LIN {X 0,Y 161.078,Z 235.028,A -85,B 0,C 180,E1 -25523.5,E2 -25523.5} C_VEL
LIN {X 0,Y 155.876,Z 225.999,A -85,B 0,C 180,E1 -25526.938,E2 -25526.938} C_VEL
LIN {X 0,Y 150.877,Z 218.256,A -85,B 0,C 180,E1 -25530.745,E2 -25530.745} C_VEL
LIN {X 0,Y 148.583,Z 214.919,A -85,B 0,C 180,E1 -25532.727,E2 -25532.727} C_VEL
LIN {X 0,Y 145.779,Z 210.989,A -85,B 0,C 180,E1 -25535.429,E2 -25535.429} C_VEL
LIN {X 0,Y 142.918,Z 207.15,A -85,B 0,C 180,E1 -25538.623,E2 -25538.623} C_VEL
LIN {X 0,Y 142.606,Z 206.481,A -85,B 0,C 180,E1 -25539.043,E2 -25539.043} C_VEL
LIN {X 0,Y 140.021,Z 203.936,A -85,B 0,C 180,E1 -25542.473,E2 -25542.473} C_VEL
LIN {X 0,Y 138.637,Z 201.246,A -85,B 0,C 180,E1 -25544.941,E2 -25544.941} C_VEL
LIN {X 0,Y 135.796,Z 198.706,A -85,B 0,C 180,E1 -25551.349,E2 -25551.349} C_VEL
LIN {X 0,Y 134.805,Z 195.544,A -85,B 0,C 180,E1 -25557.759,E2 -25557.759} C_VEL
LIN {X 0,Y 134.795,Z 195.447,A -85,B 0,C 180,E1 -25561.494,E2 -25561.494} C_VEL
LIN {X 0,Y 134.949,Z 196.715,A -85,B 0,C 180,E1 -25564.013,E2 -25564.013} C_VEL
LIN {X 0,Y 137.876,Z 200.864,A -85,B 0,C 180,E1 -25573.261,E2 -25573.261} C_VEL
LIN {X 0,Y 138.78,Z 201.463,A -85,B 0,C 180,E1 -25574.855,E2 -25574.855} C_VEL
LIN {X 0,Y 140.657,Z 204.791,A -85,B 0,C 180,E1 -25578.009,E2 -25578.009} C_VEL
LIN {X 0,Y 142.764,Z 206.915,A -85,B 0,C 180,E1 -25580.716,E2 -25580.716} C_VEL
LIN {X 0,Y 145.209,Z 210.44,A -85,B 0,C 180,E1 -25583.534,E2 -25583.534} C_VEL
LIN {X 0,Y 146.412,Z 211.841,A -85,B 0,C 180,E1 -25584.741,E2 -25584.741} C_VEL
LIN {X 0,Y 149.716,Z 216.584,A -85,B 0,C 180,E1 -25587.808,E2 -25587.808} C_VEL
LIN {X 0,Y 152.19,Z 220.352,A -85,B 0,C 180,E1 -25589.859,E2 -25589.859} C_VEL
LIN {X 0,Y 156.704,Z 229.259,A -85,B 0,C 180,E1 -25593.326,E2 -25593.326} C_VEL
LIN {X 0,Y 161.77,Z 240.791,A -85,B 0,C 180,E1 -25596.782,E2 -25596.782} C_VEL
LIN {X 0,Y 165.726,Z 251.888,A -85,B 0,C 180,E1 -25599.306,E2 -25599.306} C_VEL
LIN {X 0,Y 165.659,Z 255.549,A -85,B 0,C 180,E1 -25599.521,E2 -25599.521} C_VEL
LIN {X 0,Y 163.102,Z 287.628,A -85,B 0,C 180,E1 -25600.707,E2 -25600.707} C_VEL
LIN {X 0,Y 160.961,Z 301.09,A -85,B 0,C 180,E1 -25601.558,E2 -25601.558} C_VEL
LIN {X 0,Y 157.935,Z 313.779,A -85,B 0,C 180,E1 -25602.756,E2 -25602.756} C_VEL
LIN {X 0,Y 154.381,Z 324.846,A -85,B 0,C 180,E1 -25604.192,E2 -25604.192} C_VEL
LIN {X 0,Y 149.882,Z 336.398,A -85,B 0,C 180,E1 -25606.24,E2 -25606.24} C_VEL
LIN {X 0,Y 145.19,Z 346.81,A -85,B 0,C 180,E1 -25608.735,E2 -25608.735} C_VEL
LIN {X 0,Y 140.727,Z 355.322,A -85,B 0,C 180,E1 -25611.371,E2 -25611.371} C_VEL
LIN {X 0,Y 136.248,Z 363.183,A -85,B 0,C 180,E1 -25614.527,E2 -25614.527} C_VEL
LIN {X 0,Y 132.327,Z 369.715,A -85,B 0,C 180,E1 -25617.918,E2 -25617.918} C_VEL
LIN {X 0,Y 128.273,Z 376.146,A -85,B 0,C 180,E1 -25622.242,E2 -25622.242} C_VEL
LIN {X 0,Y 124.805,Z 381.256,A -85,B 0,C 180,E1 -25626.784,E2 -25626.784} C_VEL
LIN {X 0,Y 122.116,Z 385.23,A -85,B 0,C 180,E1 -25631.545,E2 -25631.545} C_VEL
LIN {X 0,Y 120.445,Z 388.179,A -85,B 0,C 180,E1 -25636.501,E2 -25636.501} C_VEL
LIN {X 0,Y 119.32,Z 390.59,A -85,B 0,C 180,E1 -25643.233,E2 -25643.233} C_VEL
LIN {X 0,Y 119.284,Z 391.21,A -85,B 0,C 180,E1 -25646.621,E2 -25646.621} C_VEL
LIN {X 0,Y 119.417,Z 391.429,A -85,B 0,C 180,E1 -25649.998,E2 -25649.998} C_VEL
LIN {X 0,Y 119.284,Z 391.193,A -85,B 0,C 180,E1 -25653.376,E2 -25653.376} C_VEL
LIN {X 0,Y 119.382,Z 390.566,A -85,B 0,C 180,E1 -25656.76,E2 -25656.76} C_VEL
LIN {X 0,Y 120.446,Z 388.126,A -85,B 0,C 180,E1 -25663.495,E2 -25663.495} C_VEL
LIN {X 0,Y 122.113,Z 385.154,A -85,B 0,C 180,E1 -25668.452,E2 -25668.452} C_VEL
LIN {X 0,Y 125.137,Z 380.624,A -85,B 0,C 180,E1 -25673.724,E2 -25673.724} C_VEL
LIN {X 0,Y 128.93,Z 375.007,A -85,B 0,C 180,E1 -25678.485,E2 -25678.485} C_VEL
LIN {X 0,Y 133.088,Z 368.298,A -85,B 0,C 180,E1 -25682.768,E2 -25682.768} C_VEL
LIN {X 0,Y 135.059,Z 364.976,A -85,B 0,C 180,E1 -25684.506,E2 -25684.506} C_VEL
LIN {X 0,Y 136.621,Z 361.327,A -85,B 0,C 180,E1 -25686.354,E2 -25686.354} C_VEL
LIN {X 0,Y 137.849,Z 355.051,A -85,B 0,C 180,E1 -25689.523,E2 -25689.523} C_VEL
LIN {X 0,Y 139.287,Z 348.297,A -85,B 0,C 180,E1 -25692.442,E2 -25692.442} C_VEL
LIN {X 0,Y 141.091,Z 343.81,A -85,B 0,C 180,E1 -25693.844,E2 -25693.844} C_VEL
LIN {X 0,Y 145.975,Z 333.133,A -85,B 0,C 180,E1 -25696.232,E2 -25696.232} C_VEL
LIN {X 0,Y 150.71,Z 320.63,A -85,B 0,C 180,E1 -25698.252,E2 -25698.252} C_VEL
LIN {X 0,Y 154.39,Z 308.335,A -85,B 0,C 180,E1 -25699.68,E2 -25699.68} C_VEL
LIN {X 0,Y 157.155,Z 295.303,A -85,B 0,C 180,E1 -25700.732,E2 -25700.732} C_VEL
LIN {X 0,Y 158.826,Z 282.23,A -85,B 0,C 180,E1 -25701.429,E2 -25701.429} C_VEL
LIN {X 0,Y 161.036,Z 254.175,A -85,B 0,C 180,E1 -25702.437,E2 -25702.437} C_VEL
LIN {X 0,Y 157.36,Z 243.724,A -85,B 0,C 180,E1 -25704.996,E2 -25704.996} C_VEL
LIN {X 0,Y 152.664,Z 232.741,A -85,B 0,C 180,E1 -25708.519,E2 -25708.519} C_VEL
LIN {X 0,Y 148.861,Z 224.979,A -85,B 0,C 180,E1 -25711.726,E2 -25711.726} C_VEL
LIN {X 0,Y 145.92,Z 220.592,A -85,B 0,C 180,E1 -25714.408,E2 -25714.408} C_VEL
LIN {X 0,Y 143.478,Z 217.065,A -85,B 0,C 180,E1 -25716.93,E2 -25716.93} C_VEL
LIN {X 0,Y 140.56,Z 212.9,A -85,B 0,C 180,E1 -25720.466,E2 -25720.466} C_VEL
LIN {X 0,Y 137.986,Z 209.737,A -85,B 0,C 180,E1 -25724.259,E2 -25724.259} C_VEL
LIN {X 0,Y 137.127,Z 208.03,A -85,B 0,C 180,E1 -25725.91,E2 -25725.91} C_VEL
LIN {X 0,Y 134.691,Z 205.604,A -85,B 0,C 180,E1 -25731.561,E2 -25731.561} C_VEL
LIN {X 0,Y 133.728,Z 202.571,A -85,B 0,C 180,E1 -25736.988,E2 -25736.988} C_VEL
LIN {X 0,Y 133.536,Z 202.368,A -85,B 0,C 180,E1 -25740.678,E2 -25740.678} C_VEL
LIN {X 0,Y 133.734,Z 202.746,A -85,B 0,C 180,E1 -25743.767,E2 -25743.767} C_VEL
LIN {X 0,Y 135.902,Z 207.202,A -85,B 0,C 180,E1 -25752.266,E2 -25752.266} C_VEL
LIN {X 0,Y 137.366,Z 208.395,A -85,B 0,C 180,E1 -25755.106,E2 -25755.106} C_VEL
LIN {X 0,Y 139.567,Z 211.978,A -85,B 0,C 180,E1 -25758.783,E2 -25758.783} C_VEL
LIN {X 0,Y 141.064,Z 213.572,A -85,B 0,C 180,E1 -25760.749,E2 -25760.749} C_VEL
LIN {X 0,Y 143.805,Z 217.401,A -85,B 0,C 180,E1 -25763.97,E2 -25763.97} C_VEL
LIN {X 0,Y 147.63,Z 223.134,A -85,B 0,C 180,E1 -25767.752,E2 -25767.752} C_VEL
LIN {X 0,Y 152.022,Z 230.155,A -85,B 0,C 180,E1 -25771.417,E2 -25771.417} C_VEL
LIN {X 0,Y 156.705,Z 238.412,A -85,B 0,C 180,E1 -25774.804,E2 -25774.804} C_VEL
LIN {X 0,Y 161.45,Z 247.957,A -85,B 0,C 180,E1 -25777.868,E2 -25777.868} C_VEL
LIN {X 0,Y 159.713,Z 271.663,A -85,B 0,C 180,E1 -25778.762,E2 -25778.762} C_VEL
LIN {X 0,Y 158.229,Z 285.038,A -85,B 0,C 180,E1 -25779.38,E2 -25779.38} C_VEL
LIN {X 0,Y 155.784,Z 298.21,A -85,B 0,C 180,E1 -25780.425,E2 -25780.425} C_VEL
LIN {X 0,Y 152.866,Z 309.358,A -85,B 0,C 180,E1 -25781.664,E2 -25781.664} C_VEL
LIN {X 0,Y 148.975,Z 321.287,A -85,B 0,C 180,E1 -25783.507,E2 -25783.507} C_VEL
LIN {X 0,Y 144.587,Z 331.921,A -85,B 0,C 180,E1 -25785.678,E2 -25785.678} C_VEL
LIN {X 0,Y 139.895,Z 341.613,A -85,B 0,C 180,E1 -25788.271,E2 -25788.271} C_VEL
LIN {X 0,Y 135.201,Z 350.422,A -85,B 0,C 180,E1 -25791.41,E2 -25791.41} C_VEL
LIN {X 0,Y 129.901,Z 359.017,A -85,B 0,C 180,E1 -25795.386,E2 -25795.386} C_VEL
LIN {X 0,Y 125.108,Z 365.872,A -85,B 0,C 180,E1 -25799.633,E2 -25799.633} C_VEL
LIN {X 0,Y 121.098,Z 371.353,A -85,B 0,C 180,E1 -25804.2,E2 -25804.2} C_VEL
LIN {X 0,Y 117.817,Z 375.652,A -85,B 0,C 180,E1 -25809.03,E2 -25809.03} C_VEL
LIN {X 0,Y 116.068,Z 377.924,A -85,B 0,C 180,E1 -25812.379,E2 -25812.379} C_VEL
LIN {X 0,Y 114.679,Z 379.769,A -85,B 0,C 180,E1 -25815.812,E2 -25815.812} C_VEL
LIN {X 0,Y 113.654,Z 381.152,A -85,B 0,C 180,E1 -25819.311,E2 -25819.311} C_VEL
LIN {X 0,Y 112.553,Z 382.738,A -85,B 0,C 180,E1 -25826.422,E2 -25826.422} C_VEL
LIN {X 0,Y 112.46,Z 382.938,A -85,B 0,C 180,E1 -25830.807,E2 -25830.807} C_VEL
LIN {X 0,Y 112.937,Z 382.183,A -85,B 0,C 180,E1 -25837.151,E2 -25837.151} C_VEL
LIN {X 0,Y 113.652,Z 381.217,A -85,B 0,C 180,E1 -25840.693,E2 -25840.693} C_VEL
LIN {X 0,Y 114.63,Z 379.865,A -85,B 0,C 180,E1 -25844.198,E2 -25844.198} C_VEL
LIN {X 0,Y 116.865,Z 377,A -85,B 0,C 180,E1 -25849.316,E2 -25849.316} C_VEL
LIN {X 0,Y 119.883,Z 373.112,A -85,B 0,C 180,E1 -25854.229,E2 -25854.229} C_VEL
LIN {X 0,Y 123.638,Z 368.095,A -85,B 0,C 180,E1 -25858.894,E2 -25858.894} C_VEL
LIN {X 0,Y 128.178,Z 361.767,A -85,B 0,C 180,E1 -25863.252,E2 -25863.252} C_VEL
LIN {X 0,Y 133.004,Z 354.314,A -85,B 0,C 180,E1 -25867.125,E2 -25867.125} C_VEL
LIN {X 0,Y 137.799,Z 345.963,A -85,B 0,C 180,E1 -25870.467,E2 -25870.467} C_VEL
LIN {X 0,Y 142.911,Z 335.935,A -85,B 0,C 180,E1 -25873.512,E2 -25873.512} C_VEL
LIN {X 0,Y 147.779,Z 324.829,A -85,B 0,C 180,E1 -25875.998,E2 -25875.998} C_VEL
LIN {X 0,Y 151.697,Z 313.941,A -85,B 0,C 180,E1 -25877.841,E2 -25877.841} C_VEL
LIN {X 0,Y 155.184,Z 301.895,A -85,B 0,C 180,E1 -25879.34,E2 -25879.34} C_VEL
LIN {X 0,Y 157.827,Z 288.964,A -85,B 0,C 180,E1 -25880.506,E2 -25880.506} C_VEL
LIN {X 0,Y 159.598,Z 275.623,A -85,B 0,C 180,E1 -25881.23,E2 -25881.23} C_VEL
LIN {X 0,Y 161.694,Z 248.648,A -85,B 0,C 180,E1 -25882.22,E2 -25882.22} C_VEL
LIN {X 0,Y 160.961,Z 246.685,A -85,B 0,C 180,E1 -25882.703,E2 -25882.703} C_VEL
LIN {X 0,Y 156.156,Z 237.203,A -85,B 0,C 180,E1 -25885.863,E2 -25885.863} C_VEL
LIN {X 0,Y 151.23,Z 228.617,A -85,B 0,C 180,E1 -25889.533,E2 -25889.533} C_VEL
LIN {X 0,Y 146.854,Z 221.695,A -85,B 0,C 180,E1 -25893.342,E2 -25893.342} C_VEL
LIN {X 0,Y 143.607,Z 217.135,A -85,B 0,C 180,E1 -25896.644,E2 -25896.644} C_VEL
LIN {X 0,Y 140.638,Z 212.926,A -85,B 0,C 180,E1 -25900.286,E2 -25900.286} C_VEL
LIN {X 0,Y 138.04,Z 209.692,A -85,B 0,C 180,E1 -25904.213,E2 -25904.213} C_VEL
LIN {X 0,Y 137.279,Z 208.068,A -85,B 0,C 180,E1 -25905.737,E2 -25905.737} C_VEL
LIN {X 0,Y 134.732,Z 205.56,A -85,B 0,C 180,E1 -25911.988,E2 -25911.988} C_VEL
LIN {X 0,Y 133.9,Z 202.507,A -85,B 0,C 180,E1 -25918.496,E2 -25918.496} C_VEL
LIN {X 0,Y 133.931,Z 202.725,A -85,B 0,C 180,E1 -25921.879,E2 -25921.879} C_VEL
LIN {X 0,Y 135.58,Z 206.699,A -85,B 0,C 180,E1 -25930.165,E2 -25930.165} C_VEL
LIN {X 0,Y 137.455,Z 208.381,A -85,B 0,C 180,E1 -25934.15,E2 -25934.15} C_VEL
LIN {X 0,Y 139.436,Z 211.737,A -85,B 0,C 180,E1 -25937.603,E2 -25937.603} C_VEL
LIN {X 0,Y 141.019,Z 213.431,A -85,B 0,C 180,E1 -25939.752,E2 -25939.752} C_VEL
LIN {X 0,Y 143.578,Z 217.152,A -85,B 0,C 180,E1 -25942.863,E2 -25942.863} C_VEL
LIN {X 0,Y 144.8,Z 218.877,A -85,B 0,C 180,E1 -25944.175,E2 -25944.175} C_VEL
LIN {X 0,Y 147.706,Z 223.15,A -85,B 0,C 180,E1 -25946.999,E2 -25946.999} C_VEL
LIN {X 0,Y 149.699,Z 226.419,A -85,B 0,C 180,E1 -25948.765,E2 -25948.765} C_VEL
LIN {X 0,Y 154.034,Z 235.4,A -85,B 0,C 180,E1 -25952.322,E2 -25952.322} C_VEL
LIN {X 0,Y 158.785,Z 247.167,A -85,B 0,C 180,E1 -25955.812,E2 -25955.812} C_VEL
LIN {X 0,Y 161.231,Z 254.426,A -85,B 0,C 180,E1 -25957.51,E2 -25957.51} C_VEL
LIN {X 0,Y 158.542,Z 287.605,A -85,B 0,C 180,E1 -25958.777,E2 -25958.777} C_VEL
LIN {X 0,Y 156.413,Z 300.586,A -85,B 0,C 180,E1 -25959.601,E2 -25959.601} C_VEL
LIN {X 0,Y 153.212,Z 313.527,A -85,B 0,C 180,E1 -25960.81,E2 -25960.81} C_VEL
LIN {X 0,Y 149.522,Z 324.592,A -85,B 0,C 180,E1 -25962.242,E2 -25962.242} C_VEL
LIN {X 0,Y 144.836,Z 336.143,A -85,B 0,C 180,E1 -25964.296,E2 -25964.296} C_VEL
LIN {X 0,Y 139.914,Z 346.553,A -85,B 0,C 180,E1 -25966.811,E2 -25966.811} C_VEL
LIN {X 0,Y 135.25,Z 355.066,A -85,B 0,C 180,E1 -25969.492,E2 -25969.492} C_VEL
LIN {X 0,Y 129.627,Z 364.299,A -85,B 0,C 180,E1 -25973.387,E2 -25973.387} C_VEL
LIN {X 0,Y 124.582,Z 371.977,A -85,B 0,C 180,E1 -25977.8,E2 -25977.8} C_VEL
LIN {X 0,Y 120.634,Z 377.71,A -85,B 0,C 180,E1 -25982.219,E2 -25982.219} C_VEL
LIN {X 0,Y 117.215,Z 382.434,A -85,B 0,C 180,E1 -25987.061,E2 -25987.061} C_VEL
LIN {X 0,Y 114.629,Z 386.048,A -85,B 0,C 180,E1 -25992.147,E2 -25992.147} C_VEL
LIN {X 0,Y 113.503,Z 387.919,A -85,B 0,C 180,E1 -25995.658,E2 -25995.658} C_VEL
LIN {X 0,Y 112.708,Z 389.324,A -85,B 0,C 180,E1 -25999.217,E2 -25999.217} C_VEL
LIN {X 0,Y 112.177,Z 390.95,A -85,B 0,C 180,E1 -26006.406,E2 -26006.406} C_VEL
LIN {X 0,Y 112.332,Z 391.17,A -85,B 0,C 180,E1 -26009.998,E2 -26009.998} C_VEL
LIN {X 0,Y 112.2,Z 390.934,A -85,B 0,C 180,E1 -26013.589,E2 -26013.589} C_VEL
LIN {X 0,Y 112.304,Z 390.305,A -85,B 0,C 180,E1 -26017.188,E2 -26017.188} C_VEL
LIN {X 0,Y 112.728,Z 389.287,A -85,B 0,C 180,E1 -26020.778,E2 -26020.778} C_VEL
LIN {X 0,Y 113.504,Z 387.864,A -85,B 0,C 180,E1 -26024.338,E2 -26024.338} C_VEL
LIN {X 0,Y 115.377,Z 384.893,A -85,B 0,C 180,E1 -26029.572,E2 -26029.572} C_VEL
LIN {X 0,Y 118.291,Z 380.891,A -85,B 0,C 180,E1 -26034.573,E2 -26034.573} C_VEL
LIN {X 0,Y 122.693,Z 374.745,A -85,B 0,C 180,E1 -26040.078,E2 -26040.078} C_VEL
LIN {X 0,Y 127.145,Z 368.036,A -85,B 0,C 180,E1 -26044.509,E2 -26044.509} C_VEL
LIN {X 0,Y 132.34,Z 359.723,A -85,B 0,C 180,E1 -26048.605,E2 -26048.605} C_VEL
LIN {X 0,Y 137.263,Z 351.204,A -85,B 0,C 180,E1 -26051.726,E2 -26051.726} C_VEL
LIN {X 0,Y 141.091,Z 343.81,A -85,B 0,C 180,E1 -26053.844,E2 -26053.844} C_VEL
LIN {X 0,Y 142.876,Z 339.205,A -85,B 0,C 180,E1 -26055.161,E2 -26055.161} C_VEL
LIN {X 0,Y 144.301,Z 331.465,A -85,B 0,C 180,E1 -26057.581,E2 -26057.581} C_VEL
LIN {X 0,Y 145.524,Z 323.296,A -85,B 0,C 180,E1 -26059.747,E2 -26059.747} C_VEL
LIN {X 0,Y 146.901,Z 318.027,A -85,B 0,C 180,E1 -26060.637,E2 -26060.637} C_VEL
LIN {X 0,Y 150.529,Z 305.51,A -85,B 0,C 180,E1 -26061.984,E2 -26061.984} C_VEL
LIN {X 0,Y 153.293,Z 292.019,A -85,B 0,C 180,E1 -26062.979,E2 -26062.979} C_VEL
LIN {X 0,Y 154.814,Z 278.296,A -85,B 0,C 180,E1 -26063.631,E2 -26063.631} C_VEL
LIN {X 0,Y 156.594,Z 256.462,A -85,B 0,C 180,E1 -26064.406,E2 -26064.406} C_VEL
LIN {X 0,Y 153.415,Z 247.166,A -85,B 0,C 180,E1 -26066.848,E2 -26066.848} C_VEL
LIN {X 0,Y 149.09,Z 236.597,A -85,B 0,C 180,E1 -26070.444,E2 -26070.444} C_VEL
LIN {X 0,Y 146.018,Z 230.346,A -85,B 0,C 180,E1 -26073.274,E2 -26073.274} C_VEL
LIN {X 0,Y 143.656,Z 226.611,A -85,B 0,C 180,E1 -26075.62,E2 -26075.62} C_VEL
LIN {X 0,Y 141.562,Z 223.441,A -85,B 0,C 180,E1 -26077.948,E2 -26077.948} C_VEL
LIN {X 0,Y 138.794,Z 219.375,A -85,B 0,C 180,E1 -26081.55,E2 -26081.55} C_VEL
LIN {X 0,Y 136.395,Z 216.043,A -85,B 0,C 180,E1 -26085.452,E2 -26085.452} C_VEL
LIN {X 0,Y 135.883,Z 214.882,A -85,B 0,C 180,E1 -26086.541,E2 -26086.541} C_VEL
LIN {X 0,Y 133.605,Z 212.437,A -85,B 0,C 180,E1 -26092.253,E2 -26092.253} C_VEL
LIN {X 0,Y 132.783,Z 209.548,A -85,B 0,C 180,E1 -26097.725,E2 -26097.725} C_VEL
LIN {X 0,Y 132.801,Z 209.574,A -85,B 0,C 180,E1 -26103.034,E2 -26103.034} C_VEL
LIN {X 0,Y 134.748,Z 214.068,A -85,B 0,C 180,E1 -26111.665,E2 -26111.665} C_VEL
LIN {X 0,Y 136.056,Z 215.272,A -85,B 0,C 180,E1 -26114.394,E2 -26114.394} C_VEL
LIN {X 0,Y 138.421,Z 219.021,A -85,B 0,C 180,E1 -26118.49,E2 -26118.49} C_VEL
LIN {X 0,Y 139.548,Z 220.417,A -85,B 0,C 180,E1 -26120.057,E2 -26120.057} C_VEL
LIN {X 0,Y 142.529,Z 224.85,A -85,B 0,C 180,E1 -26123.715,E2 -26123.715} C_VEL
LIN {X 0,Y 145.448,Z 229.443,A -85,B 0,C 180,E1 -26126.743,E2 -26126.743} C_VEL
LIN {X 0,Y 149.297,Z 235.841,A -85,B 0,C 180,E1 -26130.181,E2 -26130.181} C_VEL
LIN {X 0,Y 153.761,Z 244.156,A -85,B 0,C 180,E1 -26133.656,E2 -26133.656} C_VEL
LIN {X 0,Y 157.046,Z 250.976,A -85,B 0,C 180,E1 -26135.961,E2 -26135.961} C_VEL
LIN {X 0,Y 154.462,Z 280.853,A -85,B 0,C 180,E1 -26137.101,E2 -26137.101} C_VEL
LIN {X 0,Y 152.207,Z 294.25,A -85,B 0,C 180,E1 -26137.991,E2 -26137.991} C_VEL
LIN {X 0,Y 149.151,Z 306.646,A -85,B 0,C 180,E1 -26139.24,E2 -26139.24} C_VEL
LIN {X 0,Y 145.345,Z 318.414,A -85,B 0,C 180,E1 -26140.932,E2 -26140.932} C_VEL
LIN {X 0,Y 140.728,Z 329.73,A -85,B 0,C 180,E1 -26143.085,E2 -26143.085} C_VEL
LIN {X 0,Y 135.745,Z 339.925,A -85,B 0,C 180,E1 -26145.661,E2 -26145.661} C_VEL
LIN {X 0,Y 130.219,Z 349.795,A -85,B 0,C 180,E1 -26149.077,E2 -26149.077} C_VEL
LIN {X 0,Y 125.03,Z 357.954,A -85,B 0,C 180,E1 -26152.827,E2 -26152.827} C_VEL
LIN {X 0,Y 119.871,Z 365.108,A -85,B 0,C 180,E1 -26157.161,E2 -26157.161} C_VEL
LIN {X 0,Y 116.049,Z 369.93,A -85,B 0,C 180,E1 -26161.024,E2 -26161.024} C_VEL
LIN {X 0,Y 112.301,Z 374.608,A -85,B 0,C 180,E1 -26166,E2 -26166} C_VEL
LIN {X 0,Y 109.312,Z 378.185,A -85,B 0,C 180,E1 -26171.251,E2 -26171.251} C_VEL
LIN {X 0,Y 107.804,Z 380.029,A -85,B 0,C 180,E1 -26174.887,E2 -26174.887} C_VEL
LIN {X 0,Y 106.682,Z 381.411,A -85,B 0,C 180,E1 -26178.604,E2 -26178.604} C_VEL
LIN {X 0,Y 105.47,Z 382.997,A -85,B 0,C 180,E1 -26186.181,E2 -26186.181} C_VEL
LIN {X 0,Y 105.392,Z 383.22,A -85,B 0,C 180,E1 -26190.002,E2 -26190.002} C_VEL
LIN {X 0,Y 105.47,Z 383.026,A -85,B 0,C 180,E1 -26193.823,E2 -26193.823} C_VEL
LIN {X 0,Y 106.677,Z 381.476,A -85,B 0,C 180,E1 -26201.401,E2 -26201.401} C_VEL
LIN {X 0,Y 107.764,Z 380.124,A -85,B 0,C 180,E1 -26205.123,E2 -26205.123} C_VEL
LIN {X 0,Y 110.176,Z 377.259,A -85,B 0,C 180,E1 -26210.54,E2 -26210.54} C_VEL
LIN {X 0,Y 113.443,Z 373.37,A -85,B 0,C 180,E1 -26215.702,E2 -26215.702} C_VEL
LIN {X 0,Y 117.46,Z 368.353,A -85,B 0,C 180,E1 -26220.571,E2 -26220.571} C_VEL
LIN {X 0,Y 122.317,Z 362.024,A -85,B 0,C 180,E1 -26225.071,E2 -26225.071} C_VEL
LIN {X 0,Y 127.256,Z 354.816,A -85,B 0,C 180,E1 -26228.943,E2 -26228.943} C_VEL
LIN {X 0,Y 132.579,Z 346.042,A -85,B 0,C 180,E1 -26232.524,E2 -26232.524} C_VEL
LIN {X 0,Y 137.864,Z 336.19,A -85,B 0,C 180,E1 -26235.537,E2 -26235.537} C_VEL
LIN {X 0,Y 142.942,Z 325.084,A -85,B 0,C 180,E1 -26238.044,E2 -26238.044} C_VEL
LIN {X 0,Y 147.036,Z 314.194,A -85,B 0,C 180,E1 -26239.887,E2 -26239.887} C_VEL
LIN {X 0,Y 150.665,Z 302.147,A -85,B 0,C 180,E1 -26241.383,E2 -26241.383} C_VEL
LIN {X 0,Y 153.387,Z 289.445,A -85,B 0,C 180,E1 -26242.529,E2 -26242.529} C_VEL
LIN {X 0,Y 155.295,Z 275.505,A -85,B 0,C 180,E1 -26243.284,E2 -26243.284} C_VEL
LIN {X 0,Y 157.241,Z 251.093,A -85,B 0,C 180,E1 -26244.196,E2 -26244.196} C_VEL
LIN {X 0,Y 152.751,Z 241.969,A -85,B 0,C 180,E1 -26247.401,E2 -26247.401} C_VEL
LIN {X 0,Y 148.346,Z 234.012,A -85,B 0,C 180,E1 -26250.968,E2 -26250.968} C_VEL
LIN {X 0,Y 144.396,Z 227.539,A -85,B 0,C 180,E1 -26254.697,E2 -26254.697} C_VEL
LIN {X 0,Y 141.806,Z 223.606,A -85,B 0,C 180,E1 -26257.547,E2 -26257.547} C_VEL
LIN {X 0,Y 138.89,Z 219.389,A -85,B 0,C 180,E1 -26261.372,E2 -26261.372} C_VEL
LIN {X 0,Y 136.447,Z 215.964,A -85,B 0,C 180,E1 -26265.457,E2 -26265.457} C_VEL
LIN {X 0,Y 135.947,Z 214.905,A -85,B 0,C 180,E1 -26266.548,E2 -26266.548} C_VEL
LIN {X 0,Y 133.475,Z 211.92,A -85,B 0,C 180,E1 -26273.634,E2 -26273.634} C_VEL
LIN {X 0,Y 133.034,Z 209.561,A -85,B 0,C 180,E1 -26278.486,E2 -26278.486} C_VEL
LIN {X 0,Y 133.039,Z 209.652,A -85,B 0,C 180,E1 -26281.324,E2 -26281.324} C_VEL
LIN {X 0,Y 134.819,Z 214.013,A -85,B 0,C 180,E1 -26290.513,E2 -26290.513} C_VEL
LIN {X 0,Y 136.158,Z 215.239,A -85,B 0,C 180,E1 -26293.431,E2 -26293.431} C_VEL
LIN {X 0,Y 138.143,Z 218.618,A -85,B 0,C 180,E1 -26297.072,E2 -26297.072} C_VEL
LIN {X 0,Y 139.492,Z 220.252,A -85,B 0,C 180,E1 -26299.021,E2 -26299.021} C_VEL
LIN {X 0,Y 142.84,Z 225.22,A -85,B 0,C 180,E1 -26303.18,E2 -26303.18} C_VEL
LIN {X 0,Y 145.428,Z 229.244,A -85,B 0,C 180,E1 -26305.878,E2 -26305.878} C_VEL
LIN {X 0,Y 147.358,Z 232.643,A -85,B 0,C 180,E1 -26307.718,E2 -26307.718} C_VEL
LIN {X 0,Y 151.026,Z 240.853,A -85,B 0,C 180,E1 -26310.982,E2 -26310.982} C_VEL
LIN {X 0,Y 155.156,Z 251.663,A -85,B 0,C 180,E1 -26314.289,E2 -26314.289} C_VEL
LIN {X 0,Y 156.798,Z 256.709,A -85,B 0,C 180,E1 -26315.541,E2 -26315.541} C_VEL
LIN {X 0,Y 154.148,Z 287.663,A -85,B 0,C 180,E1 -26316.733,E2 -26316.733} C_VEL
LIN {X 0,Y 151.903,Z 300.766,A -85,B 0,C 180,E1 -26317.574,E2 -26317.574} C_VEL
LIN {X 0,Y 148.672,Z 313.274,A -85,B 0,C 180,E1 -26318.739,E2 -26318.739} C_VEL
LIN {X 0,Y 144.844,Z 324.338,A -85,B 0,C 180,E1 -26320.162,E2 -26320.162} C_VEL
LIN {X 0,Y 139.973,Z 335.888,A -85,B 0,C 180,E1 -26322.217,E2 -26322.217} C_VEL
LIN {X 0,Y 134.807,Z 346.296,A -85,B 0,C 180,E1 -26324.738,E2 -26324.738} C_VEL
LIN {X 0,Y 129.93,Z 354.809,A -85,B 0,C 180,E1 -26327.456,E2 -26327.456} C_VEL
LIN {X 0,Y 123.989,Z 364.042,A -85,B 0,C 180,E1 -26331.426,E2 -26331.426} C_VEL
LIN {X 0,Y 118.936,Z 371.298,A -85,B 0,C 180,E1 -26335.687,E2 -26335.687} C_VEL
LIN {X 0,Y 114.391,Z 377.452,A -85,B 0,C 180,E1 -26340.559,E2 -26340.559} C_VEL
LIN {X 0,Y 110.682,Z 382.175,A -85,B 0,C 180,E1 -26345.622,E2 -26345.622} C_VEL
LIN {X 0,Y 107.851,Z 385.788,A -85,B 0,C 180,E1 -26350.983,E2 -26350.983} C_VEL
LIN {X 0,Y 106.591,Z 387.658,A -85,B 0,C 180,E1 -26354.706,E2 -26354.706} C_VEL
LIN {X 0,Y 105.212,Z 390.072,A -85,B 0,C 180,E1 -26362.321,E2 -26362.321} C_VEL
LIN {X 0,Y 105.09,Z 390.691,A -85,B 0,C 180,E1 -26366.163,E2 -26366.163} C_VEL
LIN {X 0,Y 105.232,Z 390.911,A -85,B 0,C 180,E1 -26369.998,E2 -26369.998} C_VEL
LIN {X 0,Y 105.108,Z 390.674,A -85,B 0,C 180,E1 -26373.832,E2 -26373.832} C_VEL
LIN {X 0,Y 105.25,Z 390.045,A -85,B 0,C 180,E1 -26377.673,E2 -26377.673} C_VEL
LIN {X 0,Y 105.748,Z 389.027,A -85,B 0,C 180,E1 -26381.498,E2 -26381.498} C_VEL
LIN {X 0,Y 106.591,Z 387.602,A -85,B 0,C 180,E1 -26385.29,E2 -26385.29} C_VEL
LIN {X 0,Y 108.697,Z 384.632,A -85,B 0,C 180,E1 -26390.828,E2 -26390.828} C_VEL
LIN {X 0,Y 111.835,Z 380.629,A -85,B 0,C 180,E1 -26396.095,E2 -26396.095} C_VEL
LIN {X 0,Y 116.56,Z 374.482,A -85,B 0,C 180,E1 -26401.84,E2 -26401.84} C_VEL
LIN {X 0,Y 121.327,Z 367.773,A -85,B 0,C 180,E1 -26406.42,E2 -26406.42} C_VEL
LIN {X 0,Y 126.864,Z 359.461,A -85,B 0,C 180,E1 -26410.609,E2 -26410.609} C_VEL
LIN {X 0,Y 132.04,Z 350.941,A -85,B 0,C 180,E1 -26413.781,E2 -26413.781} C_VEL
LIN {X 0,Y 137.635,Z 340.422,A -85,B 0,C 180,E1 -26416.686,E2 -26416.686} C_VEL
LIN {X 0,Y 142.357,Z 330.013,A -85,B 0,C 180,E1 -26418.837,E2 -26418.837} C_VEL
LIN {X 0,Y 146.901,Z 318.027,A -85,B 0,C 180,E1 -26420.637,E2 -26420.637} C_VEL
LIN {X 0,Y 148.22,Z 312.667,A -85,B 0,C 180,E1 -26421.452,E2 -26421.452} C_VEL
LIN {X 0,Y 148.82,Z 303.819,A -85,B 0,C 180,E1 -26423.176,E2 -26423.176} C_VEL
LIN {X 0,Y 149.029,Z 294.775,A -85,B 0,C 180,E1 -26424.745,E2 -26424.745} C_VEL
LIN {X 0,Y 149.545,Z 289.062,A -85,B 0,C 180,E1 -26425.293,E2 -26425.293} C_VEL
LIN {X 0,Y 151.23,Z 272.24,A -85,B 0,C 180,E1 -26425.994,E2 -26425.994} C_VEL
LIN {X 0,Y 152.336,Z 258.868,A -85,B 0,C 180,E1 -26426.483,E2 -26426.483} C_VEL
LIN {X 0,Y 149.898,Z 251.421,A -85,B 0,C 180,E1 -26428.561,E2 -26428.561} C_VEL
LIN {X 0,Y 146.194,Z 241.825,A -85,B 0,C 180,E1 -26431.952,E2 -26431.952} C_VEL
LIN {X 0,Y 143.535,Z 236.081,A -85,B 0,C 180,E1 -26434.632,E2 -26434.632} C_VEL
LIN {X 0,Y 141.385,Z 232.517,A -85,B 0,C 180,E1 -26436.955,E2 -26436.955} C_VEL
LIN {X 0,Y 139.555,Z 229.618,A -85,B 0,C 180,E1 -26439.166,E2 -26439.166} C_VEL
LIN {X 0,Y 137.197,Z 225.973,A -85,B 0,C 180,E1 -26442.485,E2 -26442.485} C_VEL
LIN {X 0,Y 134.924,Z 222.474,A -85,B 0,C 180,E1 -26446.54,E2 -26446.54} C_VEL
LIN {X 0,Y 134.291,Z 221.551,A -85,B 0,C 180,E1 -26447.917,E2 -26447.917} C_VEL
LIN {X 0,Y 131.911,Z 216.995,A -85,B 0,C 180,E1 -26457.328,E2 -26457.328} C_VEL
LIN {X 0,Y 131.859,Z 216.526,A -85,B 0,C 180,E1 -26458.473,E2 -26458.473} C_VEL
LIN {X 0,Y 131.903,Z 216.732,A -85,B 0,C 180,E1 -26462.863,E2 -26462.863} C_VEL
LIN {X 0,Y 133.889,Z 221.209,A -85,B 0,C 180,E1 -26471.741,E2 -26471.741} C_VEL
LIN {X 0,Y 134.73,Z 222.028,A -85,B 0,C 180,E1 -26473.576,E2 -26473.576} C_VEL
LIN {X 0,Y 137.09,Z 225.861,A -85,B 0,C 180,E1 -26477.914,E2 -26477.914} C_VEL
LIN {X 0,Y 137.927,Z 227.056,A -85,B 0,C 180,E1 -26479.167,E2 -26479.167} C_VEL
LIN {X 0,Y 140.626,Z 231.288,A -85,B 0,C 180,E1 -26482.715,E2 -26482.715} C_VEL
LIN {X 0,Y 143.558,Z 236.091,A -85,B 0,C 180,E1 -26485.947,E2 -26485.947} C_VEL
LIN {X 0,Y 147.647,Z 243.426,A -85,B 0,C 180,E1 -26489.791,E2 -26489.791} C_VEL
LIN {X 0,Y 152.082,Z 252.369,A -85,B 0,C 180,E1 -26493.386,E2 -26493.386} C_VEL
LIN {X 0,Y 152.734,Z 253.815,A -85,B 0,C 180,E1 -26493.88,E2 -26493.88} C_VEL
LIN {X 0,Y 150.336,Z 280.898,A -85,B 0,C 180,E1 -26494.94,E2 -26494.94} C_VEL
LIN {X 0,Y 148.034,Z 294.12,A -85,B 0,C 180,E1 -26495.796,E2 -26495.796} C_VEL
LIN {X 0,Y 144.778,Z 306.911,A -85,B 0,C 180,E1 -26497.071,E2 -26497.071} C_VEL
LIN {X 0,Y 140.803,Z 318.678,A -85,B 0,C 180,E1 -26498.752,E2 -26498.752} C_VEL
LIN {X 0,Y 135.993,Z 329.992,A -85,B 0,C 180,E1 -26500.907,E2 -26500.907} C_VEL
LIN {X 0,Y 130.774,Z 340.187,A -85,B 0,C 180,E1 -26503.492,E2 -26503.492} C_VEL
LIN {X 0,Y 125.285,Z 349.494,A -85,B 0,C 180,E1 -26506.708,E2 -26506.708} C_VEL
LIN {X 0,Y 119.445,Z 358.215,A -85,B 0,C 180,E1 -26510.767,E2 -26510.767} C_VEL
LIN {X 0,Y 113.99,Z 365.368,A -85,B 0,C 180,E1 -26515.231,E2 -26515.231} C_VEL
LIN {X 0,Y 109.886,Z 370.191,A -85,B 0,C 180,E1 -26519.228,E2 -26519.228} C_VEL
LIN {X 0,Y 105.863,Z 374.868,A -85,B 0,C 180,E1 -26524.439,E2 -26524.439} C_VEL
LIN {X 0,Y 102.609,Z 378.445,A -85,B 0,C 180,E1 -26529.975,E2 -26529.975} C_VEL
LIN {X 0,Y 100.973,Z 380.289,A -85,B 0,C 180,E1 -26533.837,E2 -26533.837} C_VEL
LIN {X 0,Y 99.744,Z 381.671,A -85,B 0,C 180,E1 -26537.799,E2 -26537.799} C_VEL
LIN {X 0,Y 98.4,Z 383.256,A -85,B 0,C 180,E1 -26545.906,E2 -26545.906} C_VEL
LIN {X 0,Y 98.311,Z 383.478,A -85,B 0,C 180,E1 -26550.002,E2 -26550.002} C_VEL
LIN {X 0,Y 98.4,Z 383.284,A -85,B 0,C 180,E1 -26554.098,E2 -26554.098} C_VEL
LIN {X 0,Y 99.739,Z 381.735,A -85,B 0,C 180,E1 -26562.206,E2 -26562.206} C_VEL
LIN {X 0,Y 100.939,Z 380.382,A -85,B 0,C 180,E1 -26566.173,E2 -26566.173} C_VEL
LIN {X 0,Y 103.546,Z 377.518,A -85,B 0,C 180,E1 -26571.921,E2 -26571.921} C_VEL
LIN {X 0,Y 107.091,Z 373.628,A -85,B 0,C 180,E1 -26577.349,E2 -26577.349} C_VEL
LIN {X 0,Y 111.4,Z 368.611,A -85,B 0,C 180,E1 -26582.43,E2 -26582.43} C_VEL
LIN {X 0,Y 116.594,Z 362.28,A -85,B 0,C 180,E1 -26587.07,E2 -26587.07} C_VEL
LIN {X 0,Y 122.67,Z 353.77,A -85,B 0,C 180,E1 -26591.658,E2 -26591.658} C_VEL
LIN {X 0,Y 128.495,Z 344.524,A -85,B 0,C 180,E1 -26595.32,E2 -26595.32} C_VEL
LIN {X 0,Y 134.163,Z 334.171,A -85,B 0,C 180,E1 -26598.287,E2 -26598.287} C_VEL
LIN {X 0,Y 139.519,Z 322.495,A -85,B 0,C 180,E1 -26600.76,E2 -26600.76} C_VEL
LIN {X 0,Y 143.806,Z 310.827,A -85,B 0,C 180,E1 -26602.577,E2 -26602.577} C_VEL
LIN {X 0,Y 147.278,Z 298.68,A -85,B 0,C 180,E1 -26603.926,E2 -26603.926} C_VEL
LIN {X 0,Y 149.864,Z 285.873,A -85,B 0,C 180,E1 -26604.929,E2 -26604.929} C_VEL
LIN {X 0,Y 151.409,Z 273.497,A -85,B 0,C 180,E1 -26605.514,E2 -26605.514} C_VEL
LIN {X 0,Y 152.978,Z 254.082,A -85,B 0,C 180,E1 -26606.244,E2 -26606.244} C_VEL
LIN {X 0,Y 148.839,Z 245.469,A -85,B 0,C 180,E1 -26609.531,E2 -26609.531} C_VEL
LIN {X 0,Y 145.184,Z 238.744,A -85,B 0,C 180,E1 -26612.816,E2 -26612.816} C_VEL
LIN {X 0,Y 141.908,Z 233.174,A -85,B 0,C 180,E1 -26616.229,E2 -26616.229} C_VEL
LIN {X 0,Y 139.821,Z 229.866,A -85,B 0,C 180,E1 -26618.736,E2 -26618.736} C_VEL
LIN {X 0,Y 137.311,Z 226.007,A -85,B 0,C 180,E1 -26622.302,E2 -26622.302} C_VEL
LIN {X 0,Y 134.961,Z 222.317,A -85,B 0,C 180,E1 -26626.639,E2 -26626.639} C_VEL
LIN {X 0,Y 134.555,Z 221.688,A -85,B 0,C 180,E1 -26627.558,E2 -26627.558} C_VEL
LIN {X 0,Y 132.152,Z 216.578,A -85,B 0,C 180,E1 -26638.961,E2 -26638.961} C_VEL
LIN {X 0,Y 132.155,Z 216.649,A -85,B 0,C 180,E1 -26640.861,E2 -26640.861} C_VEL
LIN {X 0,Y 133.956,Z 221.165,A -85,B 0,C 180,E1 -26650.581,E2 -26650.581} C_VEL
LIN {X 0,Y 134.921,Z 222.194,A -85,B 0,C 180,E1 -26652.79,E2 -26652.79} C_VEL
LIN {X 0,Y 137.034,Z 225.687,A -85,B 0,C 180,E1 -26656.802,E2 -26656.802} C_VEL
LIN {X 0,Y 137.987,Z 227.073,A -85,B 0,C 180,E1 -26658.273,E2 -26658.273} C_VEL
LIN {X 0,Y 140.781,Z 231.365,A -85,B 0,C 180,E1 -26661.988,E2 -26661.988} C_VEL
LIN {X 0,Y 143.703,Z 236.179,A -85,B 0,C 180,E1 -26665.239,E2 -26665.239} C_VEL
LIN {X 0,Y 145.468,Z 239.876,A -85,B 0,C 180,E1 -26667.054,E2 -26667.054} C_VEL
LIN {X 0,Y 148.627,Z 247.619,A -85,B 0,C 180,E1 -26670.062,E2 -26670.062} C_VEL
LIN {X 0,Y 152.027,Z 257.305,A -85,B 0,C 180,E1 -26673.015,E2 -26673.015} C_VEL
LIN {X 0,Y 152.555,Z 258.958,A -85,B 0,C 180,E1 -26673.454,E2 -26673.454} C_VEL
LIN {X 0,Y 150.033,Z 287.342,A -85,B 0,C 180,E1 -26674.562,E2 -26674.562} C_VEL
LIN {X 0,Y 147.587,Z 300.945,A -85,B 0,C 180,E1 -26675.422,E2 -26675.422} C_VEL
LIN {X 0,Y 144.341,Z 313.022,A -85,B 0,C 180,E1 -26676.544,E2 -26676.544} C_VEL
LIN {X 0,Y 139.727,Z 325.668,A -85,B 0,C 180,E1 -26678.194,E2 -26678.194} C_VEL
LIN {X 0,Y 134.68,Z 336.926,A -85,B 0,C 180,E1 -26680.254,E2 -26680.254} C_VEL
LIN {X 0,Y 129.32,Z 347.072,A -85,B 0,C 180,E1 -26682.804,E2 -26682.804} C_VEL
LIN {X 0,Y 123.678,Z 356.219,A -85,B 0,C 180,E1 -26685.883,E2 -26685.883} C_VEL
LIN {X 0,Y 117.522,Z 365.145,A -85,B 0,C 180,E1 -26689.992,E2 -26689.992} C_VEL
LIN {X 0,Y 112.031,Z 372.439,A -85,B 0,C 180,E1 -26694.639,E2 -26694.639} C_VEL
LIN {X 0,Y 108.253,Z 377.194,A -85,B 0,C 180,E1 -26698.708,E2 -26698.708} C_VEL
LIN {X 0,Y 104.231,Z 381.916,A -85,B 0,C 180,E1 -26704.004,E2 -26704.004} C_VEL
LIN {X 0,Y 101.129,Z 385.528,A -85,B 0,C 180,E1 -26709.665,E2 -26709.665} C_VEL
LIN {X 0,Y 99.723,Z 387.398,A -85,B 0,C 180,E1 -26713.624,E2 -26713.624} C_VEL
LIN {X 0,Y 98.166,Z 389.812,A -85,B 0,C 180,E1 -26721.766,E2 -26721.766} C_VEL
LIN {X 0,Y 98.004,Z 390.432,A -85,B 0,C 180,E1 -26725.886,E2 -26725.886} C_VEL
LIN {X 0,Y 98.144,Z 390.652,A -85,B 0,C 180,E1 -26729.998,E2 -26729.998} C_VEL
LIN {X 0,Y 98.017,Z 390.415,A -85,B 0,C 180,E1 -26734.109,E2 -26734.109} C_VEL
LIN {X 0,Y 98.198,Z 389.785,A -85,B 0,C 180,E1 -26738.227,E2 -26738.227} C_VEL
LIN {X 0,Y 98.762,Z 388.765,A -85,B 0,C 180,E1 -26742.324,E2 -26742.324} C_VEL
LIN {X 0,Y 99.722,Z 387.341,A -85,B 0,C 180,E1 -26746.371,E2 -26746.371} C_VEL
LIN {X 0,Y 102.053,Z 384.37,A -85,B 0,C 180,E1 -26752.255,E2 -26752.255} C_VEL
LIN {X 0,Y 105.456,Z 380.367,A -85,B 0,C 180,E1 -26757.805,E2 -26757.805} C_VEL
LIN {X 0,Y 110.535,Z 374.219,A -85,B 0,C 180,E1 -26763.8,E2 -26763.8} C_VEL
LIN {X 0,Y 115.651,Z 367.51,A -85,B 0,C 180,E1 -26768.524,E2 -26768.524} C_VEL
LIN {X 0,Y 121.537,Z 359.199,A -85,B 0,C 180,E1 -26772.798,E2 -26772.798} C_VEL
LIN {X 0,Y 127.003,Z 350.679,A -85,B 0,C 180,E1 -26776,E2 -26776} C_VEL
LIN {X 0,Y 132.862,Z 340.159,A -85,B 0,C 180,E1 -26778.916,E2 -26778.916} C_VEL
LIN {X 0,Y 137.791,Z 329.75,A -85,B 0,C 180,E1 -26781.058,E2 -26781.058} C_VEL
LIN {X 0,Y 142.358,Z 318.203,A -85,B 0,C 180,E1 -26782.79,E2 -26782.79} C_VEL
LIN {X 0,Y 145.928,Z 306.544,A -85,B 0,C 180,E1 -26784.063,E2 -26784.063} C_VEL
LIN {X 0,Y 148.925,Z 292.958,A -85,B 0,C 180,E1 -26785.074,E2 -26785.074} C_VEL
LIN {X 0,Y 149.545,Z 289.062,A -85,B 0,C 180,E1 -26785.293,E2 -26785.293} C_VEL
LIN {X 0,Y 149.673,Z 285.215,A -85,B 0,C 180,E1 -26785.707,E2 -26785.707} C_VEL
LIN {X 0,Y 147.626,Z 273.272,A -85,B 0,C 180,E1 -26788.017,E2 -26788.017} C_VEL
LIN {X 0,Y 147.634,Z 269.392,A -85,B 0,C 180,E1 -26788.354,E2 -26788.354} C_VEL
LIN {X 0,Y 148.294,Z 261.229,A -85,B 0,C 180,E1 -26788.679,E2 -26788.679} C_VEL
LIN {X 0,Y 145.372,Z 252.345,A -85,B 0,C 180,E1 -26791.484,E2 -26791.484} C_VEL
LIN {X 0,Y 142.204,Z 244.049,A -85,B 0,C 180,E1 -26794.838,E2 -26794.838} C_VEL
LIN {X 0,Y 140.046,Z 239.772,A -85,B 0,C 180,E1 -26797.307,E2 -26797.307} C_VEL
LIN {X 0,Y 137.743,Z 235.968,A -85,B 0,C 180,E1 -26800.244,E2 -26800.244} C_VEL
LIN {X 0,Y 135.533,Z 232.392,A -85,B 0,C 180,E1 -26803.623,E2 -26803.623} C_VEL
LIN {X 0,Y 133.265,Z 228.543,A -85,B 0,C 180,E1 -26808.208,E2 -26808.208} C_VEL
LIN {X 0,Y 131.015,Z 224.12,A -85,B 0,C 180,E1 -26817.502,E2 -26817.502} C_VEL
LIN {X 0,Y 130.993,Z 223.588,A -85,B 0,C 180,E1 -26818.463,E2 -26818.463} C_VEL
LIN {X 0,Y 131.002,Z 223.777,A -85,B 0,C 180,E1 -26822.498,E2 -26822.498} C_VEL
LIN {X 0,Y 132.878,Z 228.201,A -85,B 0,C 180,E1 -26831.45,E2 -26831.45} C_VEL
LIN {X 0,Y 133.582,Z 229.149,A -85,B 0,C 180,E1 -26833.114,E2 -26833.114} C_VEL
LIN {X 0,Y 135.883,Z 232.811,A -85,B 0,C 180,E1 -26837.496,E2 -26837.496} C_VEL
LIN {X 0,Y 138.804,Z 237.755,A -85,B 0,C 180,E1 -26841.732,E2 -26841.732} C_VEL
LIN {X 0,Y 141.31,Z 242.098,A -85,B 0,C 180,E1 -26844.714,E2 -26844.714} C_VEL
LIN {X 0,Y 145.018,Z 249.154,A -85,B 0,C 180,E1 -26848.494,E2 -26848.494} C_VEL
LIN {X 0,Y 148.715,Z 256.974,A -85,B 0,C 180,E1 -26851.76,E2 -26851.76} C_VEL
LIN {X 0,Y 146.265,Z 281.944,A -85,B 0,C 180,E1 -26852.696,E2 -26852.696} C_VEL
LIN {X 0,Y 143.891,Z 294.939,A -85,B 0,C 180,E1 -26853.556,E2 -26853.556} C_VEL
LIN {X 0,Y 140.629,Z 307.176,A -85,B 0,C 180,E1 -26854.771,E2 -26854.771} C_VEL
LIN {X 0,Y 136.483,Z 318.942,A -85,B 0,C 180,E1 -26856.433,E2 -26856.433} C_VEL
LIN {X 0,Y 131.464,Z 330.255,A -85,B 0,C 180,E1 -26858.574,E2 -26858.574} C_VEL
LIN {X 0,Y 126.001,Z 340.449,A -85,B 0,C 180,E1 -26861.153,E2 -26861.153} C_VEL
LIN {X 0,Y 120.316,Z 349.593,A -85,B 0,C 180,E1 -26864.315,E2 -26864.315} C_VEL
LIN {X 0,Y 114.037,Z 358.477,A -85,B 0,C 180,E1 -26868.511,E2 -26868.511} C_VEL
LIN {X 0,Y 108.251,Z 365.628,A -85,B 0,C 180,E1 -26873.095,E2 -26873.095} C_VEL
LIN {X 0,Y 103.843,Z 370.452,A -85,B 0,C 180,E1 -26877.222,E2 -26877.222} C_VEL
LIN {X 0,Y 99.498,Z 375.129,A -85,B 0,C 180,E1 -26882.672,E2 -26882.672} C_VEL
LIN {X 0,Y 95.971,Z 378.705,A -85,B 0,C 180,E1 -26888.524,E2 -26888.524} C_VEL
LIN {X 0,Y 94.189,Z 380.548,A -85,B 0,C 180,E1 -26892.637,E2 -26892.637} C_VEL
LIN {X 0,Y 92.808,Z 381.931,A -85,B 0,C 180,E1 -26896.871,E2 -26896.871} C_VEL
LIN {X 0,Y 91.324,Z 383.515,A -85,B 0,C 180,E1 -26905.589,E2 -26905.589} C_VEL
LIN {X 0,Y 91.222,Z 383.737,A -85,B 0,C 180,E1 -26910.002,E2 -26910.002} C_VEL
LIN {X 0,Y 91.324,Z 383.543,A -85,B 0,C 180,E1 -26914.416,E2 -26914.416} C_VEL
LIN {X 0,Y 91.865,Z 382.958,A -85,B 0,C 180,E1 -26918.803,E2 -26918.803} C_VEL
LIN {X 0,Y 92.801,Z 381.994,A -85,B 0,C 180,E1 -26923.134,E2 -26923.134} C_VEL
LIN {X 0,Y 94.135,Z 380.641,A -85,B 0,C 180,E1 -26927.378,E2 -26927.378} C_VEL
LIN {X 0,Y 96.984,Z 377.777,A -85,B 0,C 180,E1 -26933.49,E2 -26933.49} C_VEL
LIN {X 0,Y 100.821,Z 373.887,A -85,B 0,C 180,E1 -26939.208,E2 -26939.208} C_VEL
LIN {X 0,Y 105.475,Z 368.869,A -85,B 0,C 180,E1 -26944.5,E2 -26944.5} C_VEL
LIN {X 0,Y 111.013,Z 362.537,A -85,B 0,C 180,E1 -26949.279,E2 -26949.279} C_VEL
LIN {X 0,Y 117.116,Z 354.507,A -85,B 0,C 180,E1 -26953.735,E2 -26953.735} C_VEL
LIN {X 0,Y 123.619,Z 344.779,A -85,B 0,C 180,E1 -26957.655,E2 -26957.655} C_VEL
LIN {X 0,Y 129.559,Z 334.426,A -85,B 0,C 180,E1 -26960.625,E2 -26960.625} C_VEL
LIN {X 0,Y 135.143,Z 322.749,A -85,B 0,C 180,E1 -26963.09,E2 -26963.09} C_VEL
LIN {X 0,Y 139.619,Z 311.078,A -85,B 0,C 180,E1 -26964.884,E2 -26964.884} C_VEL
LIN {X 0,Y 143.224,Z 298.93,A -85,B 0,C 180,E1 -26966.215,E2 -26966.215} C_VEL
LIN {X 0,Y 145.914,Z 286.098,A -85,B 0,C 180,E1 -26967.207,E2 -26967.207} C_VEL
LIN {X 0,Y 147.538,Z 273.436,A -85,B 0,C 180,E1 -26967.794,E2 -26967.794} C_VEL
LIN {X 0,Y 148.9,Z 257.094,A -85,B 0,C 180,E1 -26968.418,E2 -26968.418} C_VEL
LIN {X 0,Y 144.895,Z 248.588,A -85,B 0,C 180,E1 -26971.998,E2 -26971.998} C_VEL
LIN {X 0,Y 141.129,Z 241.516,A -85,B 0,C 180,E1 -26975.916,E2 -26975.916} C_VEL
LIN {X 0,Y 138.088,Z 236.315,A -85,B 0,C 180,E1 -26979.713,E2 -26979.713} C_VEL
LIN {X 0,Y 135.765,Z 232.579,A -85,B 0,C 180,E1 -26983.267,E2 -26983.267} C_VEL
LIN {X 0,Y 133.41,Z 228.578,A -85,B 0,C 180,E1 -26988.125,E2 -26988.125} C_VEL
LIN {X 0,Y 131.272,Z 223.747,A -85,B 0,C 180,E1 -26998.954,E2 -26998.954} C_VEL
LIN {X 0,Y 131.279,Z 223.644,A -85,B 0,C 180,E1 -27000.361,E2 -27000.361} C_VEL
LIN {X 0,Y 133.706,Z 229.107,A -85,B 0,C 180,E1 -27012.137,E2 -27012.137} C_VEL
LIN {X 0,Y 135.859,Z 232.676,A -85,B 0,C 180,E1 -27016.415,E2 -27016.415} C_VEL
LIN {X 0,Y 138.916,Z 237.735,A -85,B 0,C 180,E1 -27020.935,E2 -27020.935} C_VEL
LIN {X 0,Y 141.79,Z 242.712,A -85,B 0,C 180,E1 -27024.356,E2 -27024.356} C_VEL
LIN {X 0,Y 144.927,Z 250.579,A -85,B 0,C 180,E1 -27027.764,E2 -27027.764} C_VEL
LIN {X 0,Y 148.185,Z 260.289,A -85,B 0,C 180,E1 -27030.95,E2 -27030.95} C_VEL
LIN {X 0,Y 148.517,Z 261.474,A -85,B 0,C 180,E1 -27031.269,E2 -27031.269} C_VEL
LIN {X 0,Y 146.071,Z 287.414,A -85,B 0,C 180,E1 -27032.282,E2 -27032.282} C_VEL
LIN {X 0,Y 143.484,Z 301.151,A -85,B 0,C 180,E1 -27033.144,E2 -27033.144} C_VEL
LIN {X 0,Y 140.236,Z 312.769,A -85,B 0,C 180,E1 -27034.216,E2 -27034.216} C_VEL
LIN {X 0,Y 135.454,Z 325.413,A -85,B 0,C 180,E1 -27035.834,E2 -27035.834} C_VEL
LIN {X 0,Y 130.208,Z 336.671,A -85,B 0,C 180,E1 -27037.87,E2 -27037.87} C_VEL
LIN {X 0,Y 124.599,Z 346.815,A -85,B 0,C 180,E1 -27040.405,E2 -27040.405} C_VEL
LIN {X 0,Y 118.679,Z 355.962,A -85,B 0,C 180,E1 -27043.494,E2 -27043.494} C_VEL
LIN {X 0,Y 112.16,Z 364.887,A -85,B 0,C 180,E1 -27047.653,E2 -27047.653} C_VEL
LIN {X 0,Y 107.313,Z 370.961,A -85,B 0,C 180,E1 -27051.526,E2 -27051.526} C_VEL
LIN {X 0,Y 102.234,Z 376.935,A -85,B 0,C 180,E1 -27056.634,E2 -27056.634} C_VEL
LIN {X 0,Y 97.872,Z 381.656,A -85,B 0,C 180,E1 -27062.174,E2 -27062.174} C_VEL
LIN {X 0,Y 94.467,Z 385.269,A -85,B 0,C 180,E1 -27068.16,E2 -27068.16} C_VEL
LIN {X 0,Y 92.904,Z 387.138,A -85,B 0,C 180,E1 -27072.385,E2 -27072.385} C_VEL
LIN {X 0,Y 91.123,Z 389.552,A -85,B 0,C 180,E1 -27081.124,E2 -27081.124} C_VEL
LIN {X 0,Y 90.913,Z 390.172,A -85,B 0,C 180,E1 -27085.564,E2 -27085.564} C_VEL
LIN {X 0,Y 91.047,Z 390.393,A -85,B 0,C 180,E1 -27089.998,E2 -27089.998} C_VEL
LIN {X 0,Y 90.924,Z 390.155,A -85,B 0,C 180,E1 -27094.431,E2 -27094.431} C_VEL
LIN {X 0,Y 91.15,Z 389.524,A -85,B 0,C 180,E1 -27098.868,E2 -27098.868} C_VEL
LIN {X 0,Y 91.812,Z 388.505,A -85,B 0,C 180,E1 -27103.274,E2 -27103.274} C_VEL
LIN {X 0,Y 92.903,Z 387.08,A -85,B 0,C 180,E1 -27107.611,E2 -27107.611} C_VEL
LIN {X 0,Y 95.491,Z 384.109,A -85,B 0,C 180,E1 -27113.875,E2 -27113.875} C_VEL
LIN {X 0,Y 99.188,Z 380.104,A -85,B 0,C 180,E1 -27119.732,E2 -27119.732} C_VEL
LIN {X 0,Y 103.855,Z 374.963,A -85,B 0,C 180,E1 -27125.111,E2 -27125.111} C_VEL
LIN {X 0,Y 110.159,Z 367.247,A -85,B 0,C 180,E1 -27130.836,E2 -27130.836} C_VEL
LIN {X 0,Y 116.399,Z 358.936,A -85,B 0,C 180,E1 -27135.186,E2 -27135.186} C_VEL
LIN {X 0,Y 122.16,Z 350.416,A -85,B 0,C 180,E1 -27138.405,E2 -27138.405} C_VEL
LIN {X 0,Y 128.303,Z 339.896,A -85,B 0,C 180,E1 -27141.309,E2 -27141.309} C_VEL
LIN {X 0,Y 134.107,Z 328.053,A -85,B 0,C 180,E1 -27143.678,E2 -27143.678} C_VEL
LIN {X 0,Y 138.815,Z 316.111,A -85,B 0,C 180,E1 -27145.353,E2 -27145.353} C_VEL
LIN {X 0,Y 142.582,Z 303.674,A -85,B 0,C 180,E1 -27146.598,E2 -27146.598} C_VEL
LIN {X 0,Y 145.27,Z 291.076,A -85,B 0,C 180,E1 -27147.475,E2 -27147.475} C_VEL
LIN {X 0,Y 146.918,Z 276.822,A -85,B 0,C 180,E1 -27148.13,E2 -27148.13} C_VEL
LIN {X 0,Y 147.634,Z 269.392,A -85,B 0,C 180,E1 -27148.354,E2 -27148.354} C_VEL
LIN {X 0,Y 147.507,Z 266.392,A -85,B 0,C 180,E1 -27148.706,E2 -27148.706} C_VEL
LIN {X 0,Y 146.579,Z 263.364,A -85,B 0,C 180,E1 -27149.584,E2 -27149.584} C_VEL
LIN {X 0,Y 145.484,Z 261.331,A -85,B 0,C 180,E1 -27150.517,E2 -27150.517} C_VEL
LIN {X 0,Y 142.035,Z 255.835,A -85,B 0,C 180,E1 -27153.649,E2 -27153.649} C_VEL
LIN {X 0,Y 141.659,Z 254.877,A -85,B 0,C 180,E1 -27154.061,E2 -27154.061} C_VEL
LIN {X 0,Y 139.178,Z 248.198,A -85,B 0,C 180,E1 -27157.06,E2 -27157.06} C_VEL
LIN {X 0,Y 136.29,Z 242.763,A -85,B 0,C 180,E1 -27160.906,E2 -27160.906} C_VEL
LIN {X 0,Y 134.021,Z 238.978,A -85,B 0,C 180,E1 -27164.605,E2 -27164.605} C_VEL
LIN {X 0,Y 131.931,Z 235.242,A -85,B 0,C 180,E1 -27169.255,E2 -27169.255} C_VEL
LIN {X 0,Y 130.089,Z 230.589,A -85,B 0,C 180,E1 -27179.226,E2 -27179.226} C_VEL
LIN {X 0,Y 130.106,Z 230.826,A -85,B 0,C 180,E1 -27182.128,E2 -27182.128} C_VEL
LIN {X 0,Y 131.845,Z 235.163,A -85,B 0,C 180,E1 -27191.088,E2 -27191.088} C_VEL
LIN {X 0,Y 132.427,Z 236.181,A -85,B 0,C 180,E1 -27192.593,E2 -27192.593} C_VEL
LIN {X 0,Y 134.786,Z 240.237,A -85,B 0,C 180,E1 -27197.3,E2 -27197.3} C_VEL
LIN {X 0,Y 137.104,Z 244.332,A -85,B 0,C 180,E1 -27200.829,E2 -27200.829} C_VEL
LIN {X 0,Y 139.782,Z 249.332,A -85,B 0,C 180,E1 -27204.21,E2 -27204.21} C_VEL
LIN {X 0,Y 143.093,Z 256.213,A -85,B 0,C 180,E1 -27207.783,E2 -27207.783} C_VEL
LIN {X 0,Y 144.863,Z 260.2,A -85,B 0,C 180,E1 -27209.498,E2 -27209.498} C_VEL
LIN {X 0,Y 142.536,Z 282.453,A -85,B 0,C 180,E1 -27210.317,E2 -27210.317} C_VEL
LIN {X 0,Y 140.142,Z 294.99,A -85,B 0,C 180,E1 -27211.12,E2 -27211.12} C_VEL
LIN {X 0,Y 136.716,Z 307.441,A -85,B 0,C 180,E1 -27212.334,E2 -27212.334} C_VEL
LIN {X 0,Y 132.402,Z 319.205,A -85,B 0,C 180,E1 -27213.968,E2 -27213.968} C_VEL
LIN {X 0,Y 127.157,Z 330.518,A -85,B 0,C 180,E1 -27216.071,E2 -27216.071} C_VEL
LIN {X 0,Y 121.437,Z 340.712,A -85,B 0,C 180,E1 -27218.625,E2 -27218.625} C_VEL
LIN {X 0,Y 115.464,Z 349.855,A -85,B 0,C 180,E1 -27221.791,E2 -27221.791} C_VEL
LIN {X 0,Y 108.812,Z 358.738,A -85,B 0,C 180,E1 -27226.03,E2 -27226.03} C_VEL
LIN {X 0,Y 102.676,Z 365.889,A -85,B 0,C 180,E1 -27230.721,E2 -27230.721} C_VEL
LIN {X 0,Y 97.943,Z 370.713,A -85,B 0,C 180,E1 -27234.97,E2 -27234.97} C_VEL
LIN {X 0,Y 93.246,Z 375.389,A -85,B 0,C 180,E1 -27240.669,E2 -27240.669} C_VEL
LIN {X 0,Y 89.409,Z 378.965,A -85,B 0,C 180,E1 -27246.86,E2 -27246.86} C_VEL
LIN {X 0,Y 87.433,Z 380.808,A -85,B 0,C 180,E1 -27251.248,E2 -27251.248} C_VEL
LIN {X 0,Y 84.865,Z 383.172,A -85,B 0,C 180,E1 -27260.469,E2 -27260.469} C_VEL
LIN {X 0,Y 84.141,Z 383.996,A -85,B 0,C 180,E1 -27270.003,E2 -27270.003} C_VEL
LIN {X 0,Y 84.264,Z 383.802,A -85,B 0,C 180,E1 -27274.787,E2 -27274.787} C_VEL
LIN {X 0,Y 84.866,Z 383.217,A -85,B 0,C 180,E1 -27279.536,E2 -27279.536} C_VEL
LIN {X 0,Y 87.389,Z 380.899,A -85,B 0,C 180,E1 -27288.767,E2 -27288.767} C_VEL
LIN {X 0,Y 90.512,Z 378.035,A -85,B 0,C 180,E1 -27295.283,E2 -27295.283} C_VEL
LIN {X 0,Y 94.674,Z 374.146,A -85,B 0,C 180,E1 -27301.31,E2 -27301.31} C_VEL
LIN {X 0,Y 99.707,Z 369.127,A -85,B 0,C 180,E1 -27306.81,E2 -27306.81} C_VEL
LIN {X 0,Y 105.61,Z 362.795,A -85,B 0,C 180,E1 -27311.72,E2 -27311.72} C_VEL
LIN {X 0,Y 111.739,Z 355.235,A -85,B 0,C 180,E1 -27316.019,E2 -27316.019} C_VEL
LIN {X 0,Y 117.761,Z 346.811,A -85,B 0,C 180,E1 -27319.548,E2 -27319.548} C_VEL
LIN {X 0,Y 123.903,Z 336.956,A -85,B 0,C 180,E1 -27322.572,E2 -27322.572} C_VEL
LIN {X 0,Y 129.685,Z 325.847,A -85,B 0,C 180,E1 -27325.053,E2 -27325.053} C_VEL
LIN {X 0,Y 134.34,Z 314.952,A -85,B 0,C 180,E1 -27326.831,E2 -27326.831} C_VEL
LIN {X 0,Y 138.398,Z 302.901,A -85,B 0,C 180,E1 -27328.277,E2 -27328.277} C_VEL
LIN {X 0,Y 141.503,Z 289.945,A -85,B 0,C 180,E1 -27329.398,E2 -27329.398} C_VEL
LIN {X 0,Y 143.554,Z 276.702,A -85,B 0,C 180,E1 -27330.075,E2 -27330.075} C_VEL
LIN {X 0,Y 145.092,Z 260.402,A -85,B 0,C 180,E1 -27330.651,E2 -27330.651} C_VEL
LIN {X 0,Y 141.456,Z 252.375,A -85,B 0,C 180,E1 -27334.33,E2 -27334.33} C_VEL
LIN {X 0,Y 138.243,Z 246.092,A -85,B 0,C 180,E1 -27338.144,E2 -27338.144} C_VEL
LIN {X 0,Y 135.853,Z 241.927,A -85,B 0,C 180,E1 -27341.527,E2 -27341.527} C_VEL
LIN {X 0,Y 134.308,Z 239.225,A -85,B 0,C 180,E1 -27344.164,E2 -27344.164} C_VEL
LIN {X 0,Y 132.205,Z 235.39,A -85,B 0,C 180,E1 -27348.889,E2 -27348.889} C_VEL
LIN {X 0,Y 130.409,Z 230.68,A -85,B 0,C 180,E1 -27360,E2 -27360} C_VEL
LIN {X 0,Y 132.443,Z 235.832,A -85,B 0,C 180,E1 -27371.284,E2 -27371.284} C_VEL
LIN {X 0,Y 134.854,Z 240.214,A -85,B 0,C 180,E1 -27376.36,E2 -27376.36} C_VEL
LIN {X 0,Y 137.48,Z 244.777,A -85,B 0,C 180,E1 -27380.381,E2 -27380.381} C_VEL
LIN {X 0,Y 139.713,Z 249.06,A -85,B 0,C 180,E1 -27383.239,E2 -27383.239} C_VEL
LIN {X 0,Y 142.566,Z 257.012,A -85,B 0,C 180,E1 -27386.634,E2 -27386.634} C_VEL
LIN {X 0,Y 144.72,Z 263.98,A -85,B 0,C 180,E1 -27388.973,E2 -27388.973} C_VEL
LIN {X 0,Y 142.392,Z 287.256,A -85,B 0,C 180,E1 -27389.87,E2 -27389.87} C_VEL
LIN {X 0,Y 139.799,Z 300.525,A -85,B 0,C 180,E1 -27390.668,E2 -27390.668} C_VEL
LIN {X 0,Y 136.376,Z 312.517,A -85,B 0,C 180,E1 -27391.753,E2 -27391.753} C_VEL
LIN {X 0,Y 131.428,Z 325.159,A -85,B 0,C 180,E1 -27393.327,E2 -27393.327} C_VEL
LIN {X 0,Y 125.982,Z 336.417,A -85,B 0,C 180,E1 -27395.325,E2 -27395.325} C_VEL
LIN {X 0,Y 120.11,Z 346.559,A -85,B 0,C 180,E1 -27397.82,E2 -27397.82} C_VEL
LIN {X 0,Y 113.887,Z 355.704,A -85,B 0,C 180,E1 -27400.889,E2 -27400.889} C_VEL
LIN {X 0,Y 106.989,Z 364.628,A -85,B 0,C 180,E1 -27405.075,E2 -27405.075} C_VEL
LIN {X 0,Y 100.833,Z 371.815,A -85,B 0,C 180,E1 -27409.854,E2 -27409.854} C_VEL
LIN {X 0,Y 94.651,Z 378.368,A -85,B 0,C 180,E1 -27416.157,E2 -27416.157} C_VEL
LIN {X 0,Y 90.269,Z 382.708,A -85,B 0,C 180,E1 -27422.149,E2 -27422.149} C_VEL
LIN {X 0,Y 87.882,Z 385.009,A -85,B 0,C 180,E1 -27426.429,E2 -27426.429} C_VEL
LIN {X 0,Y 86.123,Z 386.878,A -85,B 0,C 180,E1 -27430.946,E2 -27430.946} C_VEL
LIN {X 0,Y 84.108,Z 389.293,A -85,B 0,C 180,E1 -27440.377,E2 -27440.377} C_VEL
LIN {X 0,Y 83.815,Z 389.913,A -85,B 0,C 180,E1 -27445.188,E2 -27445.188} C_VEL
LIN {X 0,Y 83.944,Z 390.133,A -85,B 0,C 180,E1 -27449.997,E2 -27449.997} C_VEL
LIN {X 0,Y 83.825,Z 389.895,A -85,B 0,C 180,E1 -27454.807,E2 -27454.807} C_VEL
LIN {X 0,Y 84.131,Z 389.264,A -85,B 0,C 180,E1 -27459.615,E2 -27459.615} C_VEL
LIN {X 0,Y 84.886,Z 388.244,A -85,B 0,C 180,E1 -27464.379,E2 -27464.379} C_VEL
LIN {X 0,Y 86.122,Z 386.818,A -85,B 0,C 180,E1 -27469.049,E2 -27469.049} C_VEL
LIN {X 0,Y 89.021,Z 383.848,A -85,B 0,C 180,E1 -27475.732,E2 -27475.732} C_VEL
LIN {X 0,Y 93.052,Z 379.842,A -85,B 0,C 180,E1 -27481.914,E2 -27481.914} C_VEL
LIN {X 0,Y 97.587,Z 375.238,A -85,B 0,C 180,E1 -27486.985,E2 -27486.985} C_VEL
LIN {X 0,Y 103.832,Z 368.224,A -85,B 0,C 180,E1 -27492.595,E2 -27492.595} C_VEL
LIN {X 0,Y 110.343,Z 360.166,A -85,B 0,C 180,E1 -27497.09,E2 -27497.09} C_VEL
LIN {X 0,Y 116.321,Z 351.962,A -85,B 0,C 180,E1 -27500.381,E2 -27500.381} C_VEL
LIN {X 0,Y 122.666,Z 341.96,A -85,B 0,C 180,E1 -27503.328,E2 -27503.328} C_VEL
LIN {X 0,Y 128.654,Z 330.65,A -85,B 0,C 180,E1 -27505.71,E2 -27505.71} C_VEL
LIN {X 0,Y 133.482,Z 319.571,A -85,B 0,C 180,E1 -27507.392,E2 -27507.392} C_VEL
LIN {X 0,Y 137.733,Z 307.27,A -85,B 0,C 180,E1 -27508.721,E2 -27508.721} C_VEL
LIN {X 0,Y 140.86,Z 294.519,A -85,B 0,C 180,E1 -27509.684,E2 -27509.684} C_VEL
LIN {X 0,Y 142.791,Z 281.656,A -85,B 0,C 180,E1 -27510.353,E2 -27510.353} C_VEL
LIN {X 0,Y 144.473,Z 263.674,A -85,B 0,C 180,E1 -27510.991,E2 -27510.991} C_VEL
LIN {X 0,Y 141.659,Z 254.877,A -85,B 0,C 180,E1 -27514.061,E2 -27514.061} C_VEL
LIN {X 0,Y 140.581,Z 252.496,A -85,B 0,C 180,E1 -27515.249,E2 -27515.249} C_VEL
LIN {X 0,Y 138.68,Z 250.004,A -85,B 0,C 180,E1 -27517.309,E2 -27517.309} C_VEL
LIN {X 0,Y 135.422,Z 247.688,A -85,B 0,C 180,E1 -27521.18,E2 -27521.18} C_VEL
LIN {X 0,Y 133.174,Z 246.184,A -85,B 0,C 180,E1 -27524.495,E2 -27524.495} C_VEL
LIN {X 0,Y 132.276,Z 245.127,A -85,B 0,C 180,E1 -27526.164,E2 -27526.164} C_VEL
LIN {X 0,Y 130.923,Z 242.215,A -85,B 0,C 180,E1 -27529.562,E2 -27529.562} C_VEL
LIN {X 0,Y 129.213,Z 237.884,A -85,B 0,C 180,E1 -27538.831,E2 -27538.831} C_VEL
LIN {X 0,Y 129.21,Z 237.584,A -85,B 0,C 180,E1 -27540,E2 -27540} C_VEL
LIN {X 0,Y 129.22,Z 238.106,A -85,B 0,C 180,E1 -27542.24,E2 -27542.24} C_VEL
LIN {X 0,Y 130.759,Z 242.078,A -85,B 0,C 180,E1 -27550.568,E2 -27550.568} C_VEL
LIN {X 0,Y 133.24,Z 246.75,A -85,B 0,C 180,E1 -27556.273,E2 -27556.273} C_VEL
LIN {X 0,Y 135.4,Z 250.863,A -85,B 0,C 180,E1 -27559.85,E2 -27559.85} C_VEL
LIN {X 0,Y 137.596,Z 255.263,A -85,B 0,C 180,E1 -27562.872,E2 -27562.872} C_VEL
LIN {X 0,Y 140.771,Z 262.33,A -85,B 0,C 180,E1 -27566.607,E2 -27566.607} C_VEL
LIN {X 0,Y 141.232,Z 263.417,A -85,B 0,C 180,E1 -27567.102,E2 -27567.102} C_VEL
LIN {X 0,Y 139.115,Z 282.567,A -85,B 0,C 180,E1 -27567.786,E2 -27567.786} C_VEL
LIN {X 0,Y 136.47,Z 295.964,A -85,B 0,C 180,E1 -27568.642,E2 -27568.642} C_VEL
LIN {X 0,Y 132.717,Z 308.698,A -85,B 0,C 180,E1 -27569.878,E2 -27569.878} C_VEL
LIN {X 0,Y 127.873,Z 321.047,A -85,B 0,C 180,E1 -27571.587,E2 -27571.587} C_VEL
LIN {X 0,Y 122.465,Z 332.054,A -85,B 0,C 180,E1 -27573.687,E2 -27573.687} C_VEL
LIN {X 0,Y 117.132,Z 340.975,A -85,B 0,C 180,E1 -27575.907,E2 -27575.907} C_VEL
LIN {X 0,Y 110.863,Z 350.117,A -85,B 0,C 180,E1 -27579.057,E2 -27579.057} C_VEL
LIN {X 0,Y 103.816,Z 359,A -85,B 0,C 180,E1 -27583.307,E2 -27583.307} C_VEL
LIN {X 0,Y 97.292,Z 366.149,A -85,B 0,C 180,E1 -27588.077,E2 -27588.077} C_VEL
LIN {X 0,Y 92.219,Z 370.974,A -85,B 0,C 180,E1 -27592.437,E2 -27592.437} C_VEL
LIN {X 0,Y 87.127,Z 375.649,A -85,B 0,C 180,E1 -27598.381,E2 -27598.381} C_VEL
LIN {X 0,Y 82.938,Z 379.224,A -85,B 0,C 180,E1 -27604.936,E2 -27604.936} C_VEL
LIN {X 0,Y 80.749,Z 381.068,A -85,B 0,C 180,E1 -27609.63,E2 -27609.63} C_VEL
LIN {X 0,Y 79.044,Z 382.45,A -85,B 0,C 180,E1 -27614.533,E2 -27614.533} C_VEL
LIN {X 0,Y 77.21,Z 384.033,A -85,B 0,C 180,E1 -27624.78,E2 -27624.78} C_VEL
LIN {X 0,Y 77.061,Z 384.254,A -85,B 0,C 180,E1 -27630.003,E2 -27630.003} C_VEL
LIN {X 0,Y 77.211,Z 384.06,A -85,B 0,C 180,E1 -27635.225,E2 -27635.225} C_VEL
LIN {X 0,Y 79.035,Z 382.512,A -85,B 0,C 180,E1 -27645.475,E2 -27645.475} C_VEL
LIN {X 0,Y 80.689,Z 381.158,A -85,B 0,C 180,E1 -27650.392,E2 -27650.392} C_VEL
LIN {X 0,Y 84.148,Z 378.294,A -85,B 0,C 180,E1 -27657.348,E2 -27657.348} C_VEL
LIN {X 0,Y 88.671,Z 374.405,A -85,B 0,C 180,E1 -27663.7,E2 -27663.7} C_VEL
LIN {X 0,Y 94.125,Z 369.384,A -85,B 0,C 180,E1 -27669.397,E2 -27669.397} C_VEL
LIN {X 0,Y 100.421,Z 363.052,A -85,B 0,C 180,E1 -27674.418,E2 -27674.418} C_VEL
LIN {X 0,Y 106.549,Z 355.972,A -85,B 0,C 180,E1 -27678.526,E2 -27678.526} C_VEL
LIN {X 0,Y 113.277,Z 347.068,A -85,B 0,C 180,E1 -27682.285,E2 -27682.285} C_VEL
LIN {X 0,Y 119.722,Z 337.212,A -85,B 0,C 180,E1 -27685.271,E2 -27685.271} C_VEL
LIN {X 0,Y 125.761,Z 326.101,A -85,B 0,C 180,E1 -27687.7,E2 -27687.7} C_VEL
LIN {X 0,Y 130.593,Z 315.206,A -85,B 0,C 180,E1 -27689.437,E2 -27689.437} C_VEL
LIN {X 0,Y 134.803,Z 303.153,A -85,B 0,C 180,E1 -27690.842,E2 -27690.842} C_VEL
LIN {X 0,Y 138.005,Z 290.364,A -85,B 0,C 180,E1 -27691.914,E2 -27691.914} C_VEL
LIN {X 0,Y 140.157,Z 276.932,A -85,B 0,C 180,E1 -27692.585,E2 -27692.585} C_VEL
LIN {X 0,Y 141.472,Z 263.627,A -85,B 0,C 180,E1 -27693.044,E2 -27693.044} C_VEL
LIN {X 0,Y 138.504,Z 256.891,A -85,B 0,C 180,E1 -27696.446,E2 -27696.446} C_VEL
LIN {X 0,Y 135.948,Z 251.626,A -85,B 0,C 180,E1 -27699.873,E2 -27699.873} C_VEL
LIN {X 0,Y 134.089,Z 248.141,A -85,B 0,C 180,E1 -27702.816,E2 -27702.816} C_VEL
LIN {X 0,Y 132.641,Z 245.483,A -85,B 0,C 180,E1 -27705.57,E2 -27705.57} C_VEL
LIN {X 0,Y 131.058,Z 242.231,A -85,B 0,C 180,E1 -27709.573,E2 -27709.573} C_VEL
LIN {X 0,Y 129.521,Z 237.911,A -85,B 0,C 180,E1 -27720,E2 -27720} C_VEL
LIN {X 0,Y 131.272,Z 242.718,A -85,B 0,C 180,E1 -27730.605,E2 -27730.605} C_VEL
LIN {X 0,Y 133.353,Z 246.778,A -85,B 0,C 180,E1 -27735.38,E2 -27735.38} C_VEL
LIN {X 0,Y 135.629,Z 251.035,A -85,B 0,C 180,E1 -27739.191,E2 -27739.191} C_VEL
LIN {X 0,Y 137.549,Z 255.004,A -85,B 0,C 180,E1 -27741.89,E2 -27741.89} C_VEL
LIN {X 0,Y 139.93,Z 262.506,A -85,B 0,C 180,E1 -27745.073,E2 -27745.073} C_VEL
LIN {X 0,Y 141.122,Z 266.634,A -85,B 0,C 180,E1 -27746.539,E2 -27746.539} C_VEL
LIN {X 0,Y 139.035,Z 286.808,A -85,B 0,C 180,E1 -27747.33,E2 -27747.33} C_VEL
LIN {X 0,Y 136.371,Z 300.028,A -85,B 0,C 180,E1 -27748.081,E2 -27748.081} C_VEL
LIN {X 0,Y 132.776,Z 312.264,A -85,B 0,C 180,E1 -27749.146,E2 -27749.146} C_VEL
LIN {X 0,Y 127.67,Z 324.905,A -85,B 0,C 180,E1 -27750.668,E2 -27750.668} C_VEL
LIN {X 0,Y 122.022,Z 336.162,A -85,B 0,C 180,E1 -27752.609,E2 -27752.609} C_VEL
LIN {X 0,Y 115.867,Z 346.301,A -85,B 0,C 180,E1 -27755.028,E2 -27755.028} C_VEL
LIN {X 0,Y 109.349,Z 355.446,A -85,B 0,C 180,E1 -27758.062,E2 -27758.062} C_VEL
LIN {X 0,Y 102.055,Z 364.369,A -85,B 0,C 180,E1 -27762.241,E2 -27762.241} C_VEL
LIN {X 0,Y 95.503,Z 371.557,A -85,B 0,C 180,E1 -27767.099,E2 -27767.099} C_VEL
LIN {X 0,Y 90.652,Z 376.416,A -85,B 0,C 180,E1 -27771.666,E2 -27771.666} C_VEL
LIN {X 0,Y 85.523,Z 381.138,A -85,B 0,C 180,E1 -27777.711,E2 -27777.711} C_VEL
LIN {X 0,Y 81.395,Z 384.749,A -85,B 0,C 180,E1 -27784.421,E2 -27784.421} C_VEL
LIN {X 0,Y 79.415,Z 386.618,A -85,B 0,C 180,E1 -27789.266,E2 -27789.266} C_VEL
LIN {X 0,Y 77.093,Z 389.033,A -85,B 0,C 180,E1 -27799.492,E2 -27799.492} C_VEL
LIN {X 0,Y 76.744,Z 389.654,A -85,B 0,C 180,E1 -27804.743,E2 -27804.743} C_VEL
LIN {X 0,Y 76.849,Z 389.874,A -85,B 0,C 180,E1 -27809.997,E2 -27809.997} C_VEL
LIN {X 0,Y 76.752,Z 389.635,A -85,B 0,C 180,E1 -27815.251,E2 -27815.251} C_VEL
LIN {X 0,Y 77.114,Z 389.004,A -85,B 0,C 180,E1 -27820.499,E2 -27820.499} C_VEL
LIN {X 0,Y 77.992,Z 387.983,A -85,B 0,C 180,E1 -27825.681,E2 -27825.681} C_VEL
LIN {X 0,Y 79.413,Z 386.557,A -85,B 0,C 180,E1 -27830.729,E2 -27830.729} C_VEL
LIN {X 0,Y 82.662,Z 383.587,A -85,B 0,C 180,E1 -27837.876,E2 -27837.876} C_VEL
LIN {X 0,Y 87.077,Z 379.581,A -85,B 0,C 180,E1 -27844.397,E2 -27844.397} C_VEL
LIN {X 0,Y 92.74,Z 374.153,A -85,B 0,C 180,E1 -27850.506,E2 -27850.506} C_VEL
LIN {X 0,Y 99.795,Z 366.722,A -85,B 0,C 180,E1 -27856.204,E2 -27856.204} C_VEL
LIN {X 0,Y 106.836,Z 358.411,A -85,B 0,C 180,E1 -27860.615,E2 -27860.615} C_VEL
LIN {X 0,Y 113.208,Z 349.89,A -85,B 0,C 180,E1 -27863.804,E2 -27863.804} C_VEL
LIN {X 0,Y 119.92,Z 339.369,A -85,B 0,C 180,E1 -27866.625,E2 -27866.625} C_VEL
LIN {X 0,Y 126.223,Z 327.526,A -85,B 0,C 180,E1 -27868.873,E2 -27868.873} C_VEL
LIN {X 0,Y 131.267,Z 315.58,A -85,B 0,C 180,E1 -27870.456,E2 -27870.456} C_VEL
LIN {X 0,Y 135.293,Z 303.14,A -85,B 0,C 180,E1 -27871.618,E2 -27871.618} C_VEL
LIN {X 0,Y 138.251,Z 290.023,A -85,B 0,C 180,E1 -27872.467,E2 -27872.467} C_VEL
LIN {X 0,Y 140.13,Z 274.493,A -85,B 0,C 180,E1 -27873.118,E2 -27873.118} C_VEL
LIN {X 0,Y 140.95,Z 266.558,A -85,B 0,C 180,E1 -27873.336,E2 -27873.336} C_VEL
LIN {X 0,Y 138.149,Z 257.306,A -85,B 0,C 180,E1 -27876.879,E2 -27876.879} C_VEL
LIN {X 0,Y 136.67,Z 253.392,A -85,B 0,C 180,E1 -27878.902,E2 -27878.902} C_VEL
LIN {X 0,Y 134.381,Z 248.884,A -85,B 0,C 180,E1 -27882.303,E2 -27882.303} C_VEL
LIN {X 0,Y 132.553,Z 245.535,A -85,B 0,C 180,E1 -27885.609,E2 -27885.609} C_VEL
LIN {X 0,Y 132.276,Z 245.127,A -85,B 0,C 180,E1 -27886.164,E2 -27886.164} C_VEL
LIN {X 0,Y 131.141,Z 243.863,A -85,B 0,C 180,E1 -27888.626,E2 -27888.626} C_VEL
LIN {X 0,Y 130.127,Z 243.443,A -85,B 0,C 180,E1 -27891.18,E2 -27891.18} C_VEL
LIN {X 0,Y 128.344,Z 244.639,A -85,B 0,C 180,E1 -27900.002,E2 -27900.002} C_VEL
LIN {X 0,Y 128.33,Z 245.186,A -85,B 0,C 180,E1 -27901.962,E2 -27901.962} C_VEL
LIN {X 0,Y 129.917,Z 249.549,A -85,B 0,C 180,E1 -27910.786,E2 -27910.786} C_VEL
LIN {X 0,Y 131.851,Z 253.519,A -85,B 0,C 180,E1 -27915.457,E2 -27915.457} C_VEL
LIN {X 0,Y 134.008,Z 257.911,A -85,B 0,C 180,E1 -27919.272,E2 -27919.272} C_VEL
LIN {X 0,Y 136.629,Z 263.82,A -85,B 0,C 180,E1 -27923.043,E2 -27923.043} C_VEL
LIN {X 0,Y 137.822,Z 266.828,A -85,B 0,C 180,E1 -27924.573,E2 -27924.573} C_VEL
LIN {X 0,Y 135.855,Z 283.526,A -85,B 0,C 180,E1 -27925.184,E2 -27925.184} C_VEL
LIN {X 0,Y 133.278,Z 295.951,A -85,B 0,C 180,E1 -27925.939,E2 -27925.939} C_VEL
LIN {X 0,Y 129.702,Z 307.97,A -85,B 0,C 180,E1 -27927.046,E2 -27927.046} C_VEL
LIN {X 0,Y 125.043,Z 319.732,A -85,B 0,C 180,E1 -27928.579,E2 -27928.579} C_VEL
LIN {X 0,Y 119.353,Z 331.045,A -85,B 0,C 180,E1 -27930.556,E2 -27930.556} C_VEL
LIN {X 0,Y 113.12,Z 341.237,A -85,B 0,C 180,E1 -27932.998,E2 -27932.998} C_VEL
LIN {X 0,Y 106.537,Z 350.378,A -85,B 0,C 180,E1 -27936.093,E2 -27936.093} C_VEL
LIN {X 0,Y 99.077,Z 359.262,A -85,B 0,C 180,E1 -27940.315,E2 -27940.315} C_VEL
LIN {X 0,Y 92.134,Z 366.41,A -85,B 0,C 180,E1 -27945.126,E2 -27945.126} C_VEL
LIN {X 0,Y 86.702,Z 371.234,A -85,B 0,C 180,E1 -27949.577,E2 -27949.577} C_VEL
LIN {X 0,Y 81.169,Z 375.91,A -85,B 0,C 180,E1 -27955.754,E2 -27955.754} C_VEL
LIN {X 0,Y 76.552,Z 379.485,A -85,B 0,C 180,E1 -27962.679,E2 -27962.679} C_VEL
LIN {X 0,Y 74.126,Z 381.328,A -85,B 0,C 180,E1 -27967.717,E2 -27967.717} C_VEL
LIN {X 0,Y 72.244,Z 382.709,A -85,B 0,C 180,E1 -27973.035,E2 -27973.035} C_VEL
LIN {X 0,Y 70.161,Z 384.292,A -85,B 0,C 180,E1 -27984.254,E2 -27984.254} C_VEL
LIN {X 0,Y 69.969,Z 384.513,A -85,B 0,C 180,E1 -27990.003,E2 -27990.003} C_VEL
LIN {X 0,Y 70.162,Z 384.318,A -85,B 0,C 180,E1 -27995.752,E2 -27995.752} C_VEL
LIN {X 0,Y 72.234,Z 382.77,A -85,B 0,C 180,E1 -28006.974,E2 -28006.974} C_VEL
LIN {X 0,Y 74.075,Z 381.417,A -85,B 0,C 180,E1 -28012.306,E2 -28012.306} C_VEL
LIN {X 0,Y 77.917,Z 378.552,A -85,B 0,C 180,E1 -28019.744,E2 -28019.744} C_VEL
LIN {X 0,Y 82.845,Z 374.663,A -85,B 0,C 180,E1 -28026.432,E2 -28026.432} C_VEL
LIN {X 0,Y 88.762,Z 369.641,A -85,B 0,C 180,E1 -28032.302,E2 -28032.302} C_VEL
LIN {X 0,Y 95.478,Z 363.309,A -85,B 0,C 180,E1 -28037.401,E2 -28037.401} C_VEL
LIN {X 0,Y 103.208,Z 354.783,A -85,B 0,C 180,E1 -28042.203,E2 -28042.203} C_VEL
LIN {X 0,Y 110.398,Z 345.548,A -85,B 0,C 180,E1 -28045.854,E2 -28045.854} C_VEL
LIN {X 0,Y 117.247,Z 335.189,A -85,B 0,C 180,E1 -28048.67,E2 -28048.67} C_VEL
LIN {X 0,Y 123.542,Z 323.512,A -85,B 0,C 180,E1 -28051.005,E2 -28051.005} C_VEL
LIN {X 0,Y 128.575,Z 311.835,A -85,B 0,C 180,E1 -28052.654,E2 -28052.654} C_VEL
LIN {X 0,Y 132.58,Z 299.681,A -85,B 0,C 180,E1 -28053.878,E2 -28053.878} C_VEL
LIN {X 0,Y 135.645,Z 286.475,A -85,B 0,C 180,E1 -28054.812,E2 -28054.812} C_VEL
LIN {X 0,Y 137.533,Z 272.754,A -85,B 0,C 180,E1 -28055.358,E2 -28055.358} C_VEL
LIN {X 0,Y 138.079,Z 267.025,A -85,B 0,C 180,E1 -28055.566,E2 -28055.566} C_VEL
LIN {X 0,Y 135.388,Z 260.561,A -85,B 0,C 180,E1 -28059.176,E2 -28059.176} C_VEL
LIN {X 0,Y 132.983,Z 255.461,A -85,B 0,C 180,E1 -28063.052,E2 -28063.052} C_VEL
LIN {X 0,Y 131.218,Z 251.981,A -85,B 0,C 180,E1 -28066.645,E2 -28066.645} C_VEL
LIN {X 0,Y 129.802,Z 248.959,A -85,B 0,C 180,E1 -28070.652,E2 -28070.652} C_VEL
LIN {X 0,Y 128.636,Z 245.124,A -85,B 0,C 180,E1 -28080,E2 -28080} C_VEL
LIN {X 0,Y 130.061,Z 249.461,A -85,B 0,C 180,E1 -28089.722,E2 -28089.722} C_VEL
LIN {X 0,Y 131.929,Z 253.434,A -85,B 0,C 180,E1 -28094.46,E2 -28094.46} C_VEL
LIN {X 0,Y 133.86,Z 257.318,A -85,B 0,C 180,E1 -28098.002,E2 -28098.002} C_VEL
LIN {X 0,Y 135.345,Z 260.639,A -85,B 0,C 180,E1 -28100.32,E2 -28100.32} C_VEL
LIN {X 0,Y 137.378,Z 267.748,A -85,B 0,C 180,E1 -28103.398,E2 -28103.398} C_VEL
LIN {X 0,Y 137.784,Z 269.364,A -85,B 0,C 180,E1 -28103.983,E2 -28103.983} C_VEL
LIN {X 0,Y 135.9,Z 286.752,A -85,B 0,C 180,E1 -28104.687,E2 -28104.687} C_VEL
LIN {X 0,Y 133.022,Z 300.422,A -85,B 0,C 180,E1 -28105.431,E2 -28105.431} C_VEL
LIN {X 0,Y 129.463,Z 312.011,A -85,B 0,C 180,E1 -28106.397,E2 -28106.397} C_VEL
LIN {X 0,Y 124.203,Z 324.651,A -85,B 0,C 180,E1 -28107.853,E2 -28107.853} C_VEL
LIN {X 0,Y 118.353,Z 335.907,A -85,B 0,C 180,E1 -28109.718,E2 -28109.718} C_VEL
LIN {X 0,Y 111.942,Z 346.045,A -85,B 0,C 180,E1 -28112.05,E2 -28112.05} C_VEL
LIN {X 0,Y 105.112,Z 355.189,A -85,B 0,C 180,E1 -28115.007,E2 -28115.007} C_VEL
LIN {X 0,Y 97.406,Z 364.111,A -85,B 0,C 180,E1 -28119.135,E2 -28119.135} C_VEL
LIN {X 0,Y 90.412,Z 371.298,A -85,B 0,C 180,E1 -28124.023,E2 -28124.023} C_VEL
LIN {X 0,Y 85.16,Z 376.157,A -85,B 0,C 180,E1 -28128.681,E2 -28128.681} C_VEL
LIN {X 0,Y 79.577,Z 380.878,A -85,B 0,C 180,E1 -28134.963,E2 -28134.963} C_VEL
LIN {X 0,Y 75.033,Z 384.49,A -85,B 0,C 180,E1 -28142.071,E2 -28142.071} C_VEL
LIN {X 0,Y 72.771,Z 386.358,A -85,B 0,C 180,E1 -28147.272,E2 -28147.272} C_VEL
LIN {X 0,Y 71.135,Z 387.764,A -85,B 0,C 180,E1 -28152.756,E2 -28152.756} C_VEL
LIN {X 0,Y 69.653,Z 389.394,A -85,B 0,C 180,E1 -28164.206,E2 -28164.206} C_VEL
LIN {X 0,Y 69.746,Z 389.615,A -85,B 0,C 180,E1 -28169.997,E2 -28169.997} C_VEL
LIN {X 0,Y 69.662,Z 389.375,A -85,B 0,C 180,E1 -28175.787,E2 -28175.787} C_VEL
LIN {X 0,Y 70.13,Z 388.744,A -85,B 0,C 180,E1 -28181.559,E2 -28181.559} C_VEL
LIN {X 0,Y 71.157,Z 387.722,A -85,B 0,C 180,E1 -28187.232,E2 -28187.232} C_VEL
LIN {X 0,Y 72.769,Z 386.296,A -85,B 0,C 180,E1 -28192.722,E2 -28192.722} C_VEL
LIN {X 0,Y 76.441,Z 383.326,A -85,B 0,C 180,E1 -28200.372,E2 -28200.372} C_VEL
LIN {X 0,Y 81.297,Z 379.319,A -85,B 0,C 180,E1 -28207.235,E2 -28207.235} C_VEL
LIN {X 0,Y 88.055,Z 373.299,A -85,B 0,C 180,E1 -28214.084,E2 -28214.084} C_VEL
LIN {X 0,Y 94.99,Z 366.459,A -85,B 0,C 180,E1 -28219.316,E2 -28219.316} C_VEL
LIN {X 0,Y 102.47,Z 358.149,A -85,B 0,C 180,E1 -28223.691,E2 -28223.691} C_VEL
LIN {X 0,Y 109.154,Z 349.627,A -85,B 0,C 180,E1 -28226.821,E2 -28226.821} C_VEL
LIN {X 0,Y 116.154,Z 339.105,A -85,B 0,C 180,E1 -28229.561,E2 -28229.561} C_VEL
LIN {X 0,Y 122.71,Z 327.263,A -85,B 0,C 180,E1 -28231.707,E2 -28231.707} C_VEL
LIN {X 0,Y 127.916,Z 315.314,A -85,B 0,C 180,E1 -28233.224,E2 -28233.224} C_VEL
LIN {X 0,Y 132.063,Z 302.872,A -85,B 0,C 180,E1 -28234.332,E2 -28234.332} C_VEL
LIN {X 0,Y 135.122,Z 289.743,A -85,B 0,C 180,E1 -28235.133,E2 -28235.133} C_VEL
LIN {X 0,Y 137.069,Z 274.212,A -85,B 0,C 180,E1 -28235.763,E2 -28235.763} C_VEL
LIN {X 0,Y 137.528,Z 269.142,A -85,B 0,C 180,E1 -28235.97,E2 -28235.97} C_VEL
LIN {X 0,Y 135.479,Z 261.74,A -85,B 0,C 180,E1 -28239,E2 -28239} C_VEL
LIN {X 0,Y 134.252,Z 258.362,A -85,B 0,C 180,E1 -28240.915,E2 -28240.915} C_VEL
LIN {X 0,Y 132.21,Z 254.283,A -85,B 0,C 180,E1 -28244.389,E2 -28244.389} C_VEL
LIN {X 0,Y 130.973,Z 251.828,A -85,B 0,C 180,E1 -28246.977,E2 -28246.977} C_VEL
LIN {X 0,Y 129.646,Z 248.928,A -85,B 0,C 180,E1 -28250.641,E2 -28250.641} C_VEL
LIN {X 0,Y 128.344,Z 244.639,A -85,B 0,C 180,E1 -28260.002,E2 -28260.002} C_VEL
LIN {X 0,Y 128.269,Z 245.442,A -85,B 0,C 180,E1 -28261.422,E2 -28261.422} C_VEL
LIN {X 0,Y 128.1,Z 247.958,A -85,B 0,C 180,E1 -28263.193,E2 -28263.193} C_VEL
LIN {X 0,Y 127.96,Z 253.969,A -85,B 0,C 180,E1 -28266.539,E2 -28266.539} C_VEL
LIN {X 0,Y 128.248,Z 255.411,A -85,B 0,C 180,E1 -28268.215,E2 -28268.215} C_VEL
LIN {X 0,Y 128.762,Z 256.359,A -85,B 0,C 180,E1 -28270.027,E2 -28270.027} C_VEL
LIN {X 0,Y 130.446,Z 260.191,A -85,B 0,C 180,E1 -28274.529,E2 -28274.529} C_VEL
LIN {X 0,Y 132.472,Z 264.658,A -85,B 0,C 180,E1 -28278.424,E2 -28278.424} C_VEL
LIN {X 0,Y 134.69,Z 270.273,A -85,B 0,C 180,E1 -28281.922,E2 -28281.922} C_VEL
LIN {X 0,Y 132.735,Z 285.294,A -85,B 0,C 180,E1 -28282.475,E2 -28282.475} C_VEL
LIN {X 0,Y 130.021,Z 297.48,A -85,B 0,C 180,E1 -28283.24,E2 -28283.24} C_VEL
LIN {X 0,Y 126.173,Z 309.472,A -85,B 0,C 180,E1 -28284.328,E2 -28284.328} C_VEL
LIN {X 0,Y 121.061,Z 321.574,A -85,B 0,C 180,E1 -28285.871,E2 -28285.871} C_VEL
LIN {X 0,Y 115.198,Z 332.58,A -85,B 0,C 180,E1 -28287.801,E2 -28287.801} C_VEL
LIN {X 0,Y 109.424,Z 341.498,A -85,B 0,C 180,E1 -28289.886,E2 -28289.886} C_VEL
LIN {X 0,Y 102.514,Z 350.64,A -85,B 0,C 180,E1 -28292.884,E2 -28292.884} C_VEL
LIN {X 0,Y 94.634,Z 359.523,A -85,B 0,C 180,E1 -28297.032,E2 -28297.032} C_VEL
LIN {X 0,Y 87.239,Z 366.671,A -85,B 0,C 180,E1 -28301.83,E2 -28301.83} C_VEL
LIN {X 0,Y 81.433,Z 371.495,A -85,B 0,C 180,E1 -28306.34,E2 -28306.34} C_VEL
LIN {X 0,Y 75.41,Z 376.17,A -85,B 0,C 180,E1 -28312.719,E2 -28312.719} C_VEL
LIN {X 0,Y 70.317,Z 379.745,A -85,B 0,C 180,E1 -28320.021,E2 -28320.021} C_VEL
LIN {X 0,Y 67.611,Z 381.588,A -85,B 0,C 180,E1 -28325.435,E2 -28325.435} C_VEL
LIN {X 0,Y 65.489,Z 382.969,A -85,B 0,C 180,E1 -28331.223,E2 -28331.223} C_VEL
LIN {X 0,Y 63.107,Z 384.551,A -85,B 0,C 180,E1 -28343.609,E2 -28343.609} C_VEL
LIN {X 0,Y 62.888,Z 384.772,A -85,B 0,C 180,E1 -28350.003,E2 -28350.003} C_VEL
LIN {X 0,Y 63.107,Z 384.577,A -85,B 0,C 180,E1 -28356.397,E2 -28356.397} C_VEL
LIN {X 0,Y 65.478,Z 383.028,A -85,B 0,C 180,E1 -28368.787,E2 -28368.787} C_VEL
LIN {X 0,Y 67.568,Z 381.675,A -85,B 0,C 180,E1 -28374.589,E2 -28374.589} C_VEL
LIN {X 0,Y 71.851,Z 378.81,A -85,B 0,C 180,E1 -28382.549,E2 -28382.549} C_VEL
LIN {X 0,Y 77.237,Z 374.922,A -85,B 0,C 180,E1 -28389.568,E2 -28389.568} C_VEL
LIN {X 0,Y 83.658,Z 369.899,A -85,B 0,C 180,E1 -28395.57,E2 -28395.57} C_VEL
LIN {X 0,Y 90.822,Z 363.567,A -85,B 0,C 180,E1 -28400.701,E2 -28400.701} C_VEL
LIN {X 0,Y 98.515,Z 355.593,A -85,B 0,C 180,E1 -28405.199,E2 -28405.199} C_VEL
LIN {X 0,Y 106.58,Z 345.804,A -85,B 0,C 180,E1 -28409.01,E2 -28409.01} C_VEL
LIN {X 0,Y 113.726,Z 335.444,A -85,B 0,C 180,E1 -28411.719,E2 -28411.719} C_VEL
LIN {X 0,Y 120.273,Z 323.766,A -85,B 0,C 180,E1 -28413.954,E2 -28413.954} C_VEL
LIN {X 0,Y 125.479,Z 312.088,A -85,B 0,C 180,E1 -28415.528,E2 -28415.528} C_VEL
LIN {X 0,Y 129.678,Z 299.743,A -85,B 0,C 180,E1 -28416.7,E2 -28416.7} C_VEL
LIN {X 0,Y 132.85,Z 286.401,A -85,B 0,C 180,E1 -28417.596,E2 -28417.596} C_VEL
LIN {X 0,Y 134.734,Z 272.99,A -85,B 0,C 180,E1 -28418.097,E2 -28418.097} C_VEL
LIN {X 0,Y 134.937,Z 270.428,A -85,B 0,C 180,E1 -28418.242,E2 -28418.242} C_VEL
LIN {X 0,Y 132.561,Z 264.443,A -85,B 0,C 180,E1 -28422.033,E2 -28422.033} C_VEL
LIN {X 0,Y 130.331,Z 259.411,A -85,B 0,C 180,E1 -28426.552,E2 -28426.552} C_VEL
LIN {X 0,Y 128.676,Z 255.775,A -85,B 0,C 180,E1 -28431.46,E2 -28431.46} C_VEL
LIN {X 0,Y 127.749,Z 252.343,A -85,B 0,C 180,E1 -28440,E2 -28440} C_VEL
LIN {X 0,Y 128.936,Z 256.326,A -85,B 0,C 180,E1 -28449.016,E2 -28449.016} C_VEL
LIN {X 0,Y 130.544,Z 260.081,A -85,B 0,C 180,E1 -28453.524,E2 -28453.524} C_VEL
LIN {X 0,Y 132.386,Z 264.093,A -85,B 0,C 180,E1 -28457.198,E2 -28457.198} C_VEL
LIN {X 0,Y 133.42,Z 266.947,A -85,B 0,C 180,E1 -28459.022,E2 -28459.022} C_VEL
LIN {X 0,Y 134.732,Z 272.171,A -85,B 0,C 180,E1 -28461.316,E2 -28461.316} C_VEL
LIN {X 0,Y 133.019,Z 286.948,A -85,B 0,C 180,E1 -28461.93,E2 -28461.93} C_VEL
LIN {X 0,Y 130.024,Z 300.576,A -85,B 0,C 180,E1 -28462.628,E2 -28462.628} C_VEL
LIN {X 0,Y 126.466,Z 311.758,A -85,B 0,C 180,E1 -28463.515,E2 -28463.515} C_VEL
LIN {X 0,Y 121.053,Z 324.398,A -85,B 0,C 180,E1 -28464.884,E2 -28464.884} C_VEL
LIN {X 0,Y 114.999,Z 335.652,A -85,B 0,C 180,E1 -28466.645,E2 -28466.645} C_VEL
LIN {X 0,Y 108.346,Z 345.789,A -85,B 0,C 180,E1 -28468.871,E2 -28468.871} C_VEL
LIN {X 0,Y 101.204,Z 354.932,A -85,B 0,C 180,E1 -28471.711,E2 -28471.711} C_VEL
LIN {X 0,Y 93.063,Z 363.853,A -85,B 0,C 180,E1 -28475.723,E2 -28475.723} C_VEL
LIN {X 0,Y 85.604,Z 371.039,A -85,B 0,C 180,E1 -28480.584,E2 -28480.584} C_VEL
LIN {X 0,Y 79.914,Z 375.896,A -85,B 0,C 180,E1 -28485.284,E2 -28485.284} C_VEL
LIN {X 0,Y 73.835,Z 380.618,A -85,B 0,C 180,E1 -28491.776,E2 -28491.776} C_VEL
LIN {X 0,Y 68.825,Z 384.231,A -85,B 0,C 180,E1 -28499.295,E2 -28499.295} C_VEL
LIN {X 0,Y 66.235,Z 386.098,A -85,B 0,C 180,E1 -28504.883,E2 -28504.883} C_VEL
LIN {X 0,Y 64.359,Z 387.504,A -85,B 0,C 180,E1 -28510.874,E2 -28510.874} C_VEL
LIN {X 0,Y 62.576,Z 389.134,A -85,B 0,C 180,E1 -28523.548,E2 -28523.548} C_VEL
LIN {X 0,Y 62.665,Z 389.356,A -85,B 0,C 180,E1 -28529.997,E2 -28529.997} C_VEL
LIN {X 0,Y 62.586,Z 389.115,A -85,B 0,C 180,E1 -28536.444,E2 -28536.444} C_VEL
LIN {X 0,Y 63.163,Z 388.483,A -85,B 0,C 180,E1 -28542.854,E2 -28542.854} C_VEL
LIN {X 0,Y 64.375,Z 387.461,A -85,B 0,C 180,E1 -28549.114,E2 -28549.114} C_VEL
LIN {X 0,Y 66.233,Z 386.034,A -85,B 0,C 180,E1 -28555.111,E2 -28555.111} C_VEL
LIN {X 0,Y 70.395,Z 383.066,A -85,B 0,C 180,E1 -28563.301,E2 -28563.301} C_VEL
LIN {X 0,Y 75.75,Z 379.058,A -85,B 0,C 180,E1 -28570.496,E2 -28570.496} C_VEL
LIN {X 0,Y 82.571,Z 373.493,A -85,B 0,C 180,E1 -28577.085,E2 -28577.085} C_VEL
LIN {X 0,Y 90.505,Z 366.197,A -85,B 0,C 180,E1 -28582.739,E2 -28582.739} C_VEL
LIN {X 0,Y 98.427,Z 357.887,A -85,B 0,C 180,E1 -28587.028,E2 -28587.028} C_VEL
LIN {X 0,Y 105.425,Z 349.364,A -85,B 0,C 180,E1 -28590.063,E2 -28590.063} C_VEL
LIN {X 0,Y 112.728,Z 338.842,A -85,B 0,C 180,E1 -28592.669,E2 -28592.669} C_VEL
LIN {X 0,Y 118.747,Z 328.432,A -85,B 0,C 180,E1 -28594.491,E2 -28594.491} C_VEL
LIN {X 0,Y 124.096,Z 317.006,A -85,B 0,C 180,E1 -28595.947,E2 -28595.947} C_VEL
LIN {X 0,Y 128.357,Z 305.22,A -85,B 0,C 180,E1 -28596.995,E2 -28596.995} C_VEL
LIN {X 0,Y 131.707,Z 292.314,A -85,B 0,C 180,E1 -28597.787,E2 -28597.787} C_VEL
LIN {X 0,Y 133.723,Z 279.395,A -85,B 0,C 180,E1 -28598.369,E2 -28598.369} C_VEL
LIN {X 0,Y 134.469,Z 271.934,A -85,B 0,C 180,E1 -28598.638,E2 -28598.638} C_VEL
LIN {X 0,Y 132.842,Z 265.632,A -85,B 0,C 180,E1 -28601.493,E2 -28601.493} C_VEL
LIN {X 0,Y 131.008,Z 261.406,A -85,B 0,C 180,E1 -28604.845,E2 -28604.845} C_VEL
LIN {X 0,Y 129.591,Z 258.347,A -85,B 0,C 180,E1 -28608.068,E2 -28608.068} C_VEL
LIN {X 0,Y 128.529,Z 255.798,A -85,B 0,C 180,E1 -28611.352,E2 -28611.352} C_VEL
LIN {X 0,Y 127.475,Z 251.715,A -85,B 0,C 180,E1 -28620,E2 -28620} C_VEL
LIN {X 0,Y 127.444,Z 252.31,A -85,B 0,C 180,E1 -28621.778,E2 -28621.778} C_VEL
LIN {X 0,Y 128.248,Z 255.411,A -85,B 0,C 180,E1 -28628.215,E2 -28628.215} C_VEL
LIN {X 0,Y 128.621,Z 256.85,A -85,B 0,C 180,E1 -28629.818,E2 -28629.818} C_VEL
LIN {X 0,Y 128.867,Z 259.343,A -85,B 0,C 180,E1 -28631.192,E2 -28631.192} C_VEL
LIN {X 0,Y 129.542,Z 267.317,A -85,B 0,C 180,E1 -28634.526,E2 -28634.526} C_VEL
LIN {X 0,Y 129.93,Z 268.87,A -85,B 0,C 180,E1 -28635.509,E2 -28635.509} C_VEL
LIN {X 0,Y 131.623,Z 273.355,A -85,B 0,C 180,E1 -28638.786,E2 -28638.786} C_VEL
LIN {X 0,Y 131.833,Z 273.948,A -85,B 0,C 180,E1 -28639.155,E2 -28639.155} C_VEL
LIN {X 0,Y 129.774,Z 287.724,A -85,B 0,C 180,E1 -28639.701,E2 -28639.701} C_VEL
LIN {X 0,Y 126.77,Z 299.867,A -85,B 0,C 180,E1 -28640.484,E2 -28640.484} C_VEL
LIN {X 0,Y 122.6,Z 311.879,A -85,B 0,C 180,E1 -28641.562,E2 -28641.562} C_VEL
LIN {X 0,Y 117.388,Z 323.395,A -85,B 0,C 180,E1 -28643.007,E2 -28643.007} C_VEL
LIN {X 0,Y 111.318,Z 334.02,A -85,B 0,C 180,E1 -28644.836,E2 -28644.836} C_VEL
LIN {X 0,Y 104.603,Z 343.71,A -85,B 0,C 180,E1 -28647.104,E2 -28647.104} C_VEL
LIN {X 0,Y 97.437,Z 352.52,A -85,B 0,C 180,E1 -28650.061,E2 -28650.061} C_VEL
LIN {X 0,Y 89.223,Z 361.105,A -85,B 0,C 180,E1 -28654.206,E2 -28654.206} C_VEL
LIN {X 0,Y 81.399,Z 367.955,A -85,B 0,C 180,E1 -28659.013,E2 -28659.013} C_VEL
LIN {X 0,Y 74.166,Z 373.439,A -85,B 0,C 180,E1 -28664.713,E2 -28664.713} C_VEL
LIN {X 0,Y 67.896,Z 377.733,A -85,B 0,C 180,E1 -28671.611,E2 -28671.611} C_VEL
LIN {X 0,Y 64.269,Z 380.005,A -85,B 0,C 180,E1 -28676.859,E2 -28676.859} C_VEL
LIN {X 0,Y 61.233,Z 381.847,A -85,B 0,C 180,E1 -28682.675,E2 -28682.675} C_VEL
LIN {X 0,Y 57.086,Z 384.209,A -85,B 0,C 180,E1 -28695.75,E2 -28695.75} C_VEL
LIN {X 0,Y 56.082,Z 384.809,A -85,B 0,C 180,E1 -28702.805,E2 -28702.805} C_VEL
LIN {X 0,Y 55.809,Z 385.03,A -85,B 0,C 180,E1 -28710.004,E2 -28710.004} C_VEL
LIN {X 0,Y 56.083,Z 384.835,A -85,B 0,C 180,E1 -28717.203,E2 -28717.203} C_VEL
LIN {X 0,Y 58.796,Z 383.287,A -85,B 0,C 180,E1 -28731.018,E2 -28731.018} C_VEL
LIN {X 0,Y 61.197,Z 381.933,A -85,B 0,C 180,E1 -28737.35,E2 -28737.35} C_VEL
LIN {X 0,Y 65.973,Z 379.068,A -85,B 0,C 180,E1 -28745.87,E2 -28745.87} C_VEL
LIN {X 0,Y 71.897,Z 375.18,A -85,B 0,C 180,E1 -28753.18,E2 -28753.18} C_VEL
LIN {X 0,Y 78.861,Z 370.156,A -85,B 0,C 180,E1 -28759.248,E2 -28759.248} C_VEL
LIN {X 0,Y 86.5,Z 363.824,A -85,B 0,C 180,E1 -28764.342,E2 -28764.342} C_VEL
LIN {X 0,Y 94.112,Z 356.41,A -85,B 0,C 180,E1 -28768.484,E2 -28768.484} C_VEL
LIN {X 0,Y 101.665,Z 347.836,A -85,B 0,C 180,E1 -28771.814,E2 -28771.814} C_VEL
LIN {X 0,Y 109.027,Z 337.977,A -85,B 0,C 180,E1 -28774.485,E2 -28774.485} C_VEL
LIN {X 0,Y 115.809,Z 326.863,A -85,B 0,C 180,E1 -28776.62,E2 -28776.62} C_VEL
LIN {X 0,Y 121.184,Z 315.964,A -85,B 0,C 180,E1 -28778.114,E2 -28778.114} C_VEL
LIN {X 0,Y 125.944,Z 303.563,A -85,B 0,C 180,E1 -28779.353,E2 -28779.353} C_VEL
LIN {X 0,Y 129.439,Z 290.774,A -85,B 0,C 180,E1 -28780.261,E2 -28780.261} C_VEL
LIN {X 0,Y 131.809,Z 277.049,A -85,B 0,C 180,E1 -28780.835,E2 -28780.835} C_VEL
LIN {X 0,Y 132.091,Z 274.117,A -85,B 0,C 180,E1 -28781.007,E2 -28781.007} C_VEL
LIN {X 0,Y 130.561,Z 270.019,A -85,B 0,C 180,E1 -28783.885,E2 -28783.885} C_VEL
LIN {X 0,Y 128.891,Z 265.839,A -85,B 0,C 180,E1 -28787.802,E2 -28787.802} C_VEL
LIN {X 0,Y 127.626,Z 262.663,A -85,B 0,C 180,E1 -28792.087,E2 -28792.087} C_VEL
LIN {X 0,Y 126.868,Z 259.521,A -85,B 0,C 180,E1 -28800,E2 -28800} C_VEL
LIN {X 0,Y 127.863,Z 263.309,A -85,B 0,C 180,E1 -28808.436,E2 -28808.436} C_VEL
LIN {X 0,Y 129.193,Z 266.729,A -85,B 0,C 180,E1 -28812.568,E2 -28812.568} C_VEL
LIN {X 0,Y 130.95,Z 270.959,A -85,B 0,C 180,E1 -28816.412,E2 -28816.412} C_VEL
LIN {X 0,Y 132.014,Z 275.343,A -85,B 0,C 180,E1 -28818.628,E2 -28818.628} C_VEL
LIN {X 0,Y 129.989,Z 289.779,A -85,B 0,C 180,E1 -28819.156,E2 -28819.156} C_VEL
LIN {X 0,Y 126.98,Z 301.964,A -85,B 0,C 180,E1 -28819.793,E2 -28819.793} C_VEL
LIN {X 0,Y 122.951,Z 313.62,A -85,B 0,C 180,E1 -28820.676,E2 -28820.676} C_VEL
LIN {X 0,Y 117.46,Z 325.728,A -85,B 0,C 180,E1 -28821.962,E2 -28821.962} C_VEL
LIN {X 0,Y 111.208,Z 336.638,A -85,B 0,C 180,E1 -28823.599,E2 -28823.599} C_VEL
LIN {X 0,Y 103.586,Z 347.488,A -85,B 0,C 180,E1 -28825.974,E2 -28825.974} C_VEL
LIN {X 0,Y 96.196,Z 356.309,A -85,B 0,C 180,E1 -28828.749,E2 -28828.749} C_VEL
LIN {X 0,Y 89.095,Z 363.595,A -85,B 0,C 180,E1 -28832.004,E2 -28832.004} C_VEL
LIN {X 0,Y 81.143,Z 370.78,A -85,B 0,C 180,E1 -28836.755,E2 -28836.755} C_VEL
LIN {X 0,Y 74.972,Z 375.635,A -85,B 0,C 180,E1 -28841.412,E2 -28841.412} C_VEL
LIN {X 0,Y 68.365,Z 380.359,A -85,B 0,C 180,E1 -28848.068,E2 -28848.068} C_VEL
LIN {X 0,Y 62.815,Z 383.972,A -85,B 0,C 180,E1 -28855.981,E2 -28855.981} C_VEL
LIN {X 0,Y 59.843,Z 385.837,A -85,B 0,C 180,E1 -28861.978,E2 -28861.978} C_VEL
LIN {X 0,Y 56.219,Z 388.254,A -85,B 0,C 180,E1 -28875.518,E2 -28875.518} C_VEL
LIN {X 0,Y 55.525,Z 388.875,A -85,B 0,C 180,E1 -28882.725,E2 -28882.725} C_VEL
LIN {X 0,Y 55.573,Z 389.097,A -85,B 0,C 180,E1 -28889.996,E2 -28889.996} C_VEL
LIN {X 0,Y 55.534,Z 388.855,A -85,B 0,C 180,E1 -28897.266,E2 -28897.266} C_VEL
LIN {X 0,Y 56.247,Z 388.223,A -85,B 0,C 180,E1 -28904.467,E2 -28904.467} C_VEL
LIN {X 0,Y 57.666,Z 387.2,A -85,B 0,C 180,E1 -28911.442,E2 -28911.442} C_VEL
LIN {X 0,Y 59.841,Z 385.772,A -85,B 0,C 180,E1 -28918.016,E2 -28918.016} C_VEL
LIN {X 0,Y 64.545,Z 382.804,A -85,B 0,C 180,E1 -28926.784,E2 -28926.784} C_VEL
LIN {X 0,Y 70.49,Z 378.797,A -85,B 0,C 180,E1 -28934.255,E2 -28934.255} C_VEL
LIN {X 0,Y 78.582,Z 372.675,A -85,B 0,C 180,E1 -28941.426,E2 -28941.426} C_VEL
LIN {X 0,Y 86.366,Z 365.934,A -85,B 0,C 180,E1 -28946.515,E2 -28946.515} C_VEL
LIN {X 0,Y 94.737,Z 357.624,A -85,B 0,C 180,E1 -28950.646,E2 -28950.646} C_VEL
LIN {X 0,Y 102.058,Z 349.101,A -85,B 0,C 180,E1 -28953.529,E2 -28953.529} C_VEL
LIN {X 0,Y 109.648,Z 338.579,A -85,B 0,C 180,E1 -28955.968,E2 -28955.968} C_VEL
LIN {X 0,Y 115.873,Z 328.169,A -85,B 0,C 180,E1 -28957.654,E2 -28957.654} C_VEL
LIN {X 0,Y 121.329,Z 316.848,A -85,B 0,C 180,E1 -28958.997,E2 -28958.997} C_VEL
LIN {X 0,Y 125.623,Z 305.376,A -85,B 0,C 180,E1 -28959.945,E2 -28959.945} C_VEL
LIN {X 0,Y 129.166,Z 292.146,A -85,B 0,C 180,E1 -28960.7,E2 -28960.7} C_VEL
LIN {X 0,Y 131.336,Z 278.565,A -85,B 0,C 180,E1 -28961.273,E2 -28961.273} C_VEL
LIN {X 0,Y 131.695,Z 274.877,A -85,B 0,C 180,E1 -28961.426,E2 -28961.426} C_VEL
LIN {X 0,Y 130.646,Z 270.668,A -85,B 0,C 180,E1 -28963.595,E2 -28963.595} C_VEL
LIN {X 0,Y 128.988,Z 266.583,A -85,B 0,C 180,E1 -28967.212,E2 -28967.212} C_VEL
LIN {X 0,Y 127.384,Z 262.559,A -85,B 0,C 180,E1 -28972.272,E2 -28972.272} C_VEL
LIN {X 0,Y 126.581,Z 258.994,A -85,B 0,C 180,E1 -28980,E2 -28980} C_VEL
LIN {X 0,Y 126.561,Z 259.29,A -85,B 0,C 180,E1 -28981.252,E2 -28981.252} C_VEL
LIN {X 0,Y 127.642,Z 263.22,A -85,B 0,C 180,E1 -28989.308,E2 -28989.308} C_VEL
LIN {X 0,Y 129.12,Z 266.915,A -85,B 0,C 180,E1 -28993.676,E2 -28993.676} C_VEL
LIN {X 0,Y 129.93,Z 268.87,A -85,B 0,C 180,E1 -28995.509,E2 -28995.509} C_VEL
LIN {X 0,Y 130.211,Z 270.568,A -85,B 0,C 180,E1 -28996.285,E2 -28996.285} C_VEL
LIN {X 0,Y 130.176,Z 274.116,A -85,B 0,C 180,E1 -28996.911,E2 -28996.911} C_VEL
LIN {X 0,Y 129.705,Z 278.037,A -85,B 0,C 180,E1 -28997.051,E2 -28997.051} C_VEL
LIN {X 0,Y 127.485,Z 288.332,A -85,B 0,C 180,E1 -28996.709,E2 -28996.709} C_VEL
LIN {X 0,Y 127.165,Z 289.794,A -85,B 0,C 180,E1 -28996.789,E2 -28996.789} C_VEL
LIN {X 0,Y 123.631,Z 302.863,A -85,B 0,C 180,E1 -28997.625,E2 -28997.625} C_VEL
LIN {X 0,Y 118.729,Z 315.466,A -85,B 0,C 180,E1 -28998.728,E2 -28998.728} C_VEL
LIN {X 0,Y 113.226,Z 326.509,A -85,B 0,C 180,E1 -29000.154,E2 -29000.154} C_VEL
LIN {X 0,Y 106.191,Z 337.771,A -85,B 0,C 180,E1 -29002.103,E2 -29002.103} C_VEL
LIN {X 0,Y 98.544,Z 347.71,A -85,B 0,C 180,E1 -29004.596,E2 -29004.596} C_VEL
LIN {X 0,Y 91.256,Z 355.75,A -85,B 0,C 180,E1 -29007.522,E2 -29007.522} C_VEL
LIN {X 0,Y 82.6,Z 363.816,A -85,B 0,C 180,E1 -29011.702,E2 -29011.702} C_VEL
LIN {X 0,Y 74.469,Z 370.21,A -85,B 0,C 180,E1 -29016.666,E2 -29016.666} C_VEL
LIN {X 0,Y 66.936,Z 375.281,A -85,B 0,C 180,E1 -29022.701,E2 -29022.701} C_VEL
LIN {X 0,Y 60.406,Z 379.209,A -85,B 0,C 180,E1 -29030.22,E2 -29030.22} C_VEL
LIN {X 0,Y 55.011,Z 382.108,A -85,B 0,C 180,E1 -29039.273,E2 -29039.273} C_VEL
LIN {X 0,Y 52.247,Z 383.488,A -85,B 0,C 180,E1 -29046.205,E2 -29046.205} C_VEL
LIN {X 0,Y 49.061,Z 385.068,A -85,B 0,C 180,E1 -29061.768,E2 -29061.768} C_VEL
LIN {X 0,Y 48.73,Z 385.289,A -85,B 0,C 180,E1 -29070.004,E2 -29070.004} C_VEL
LIN {X 0,Y 49.061,Z 385.094,A -85,B 0,C 180,E1 -29078.24,E2 -29078.24} C_VEL
LIN {X 0,Y 52.238,Z 383.546,A -85,B 0,C 180,E1 -29093.809,E2 -29093.809} C_VEL
LIN {X 0,Y 54.978,Z 382.192,A -85,B 0,C 180,E1 -29100.757,E2 -29100.757} C_VEL
LIN {X 0,Y 60.367,Z 379.326,A -85,B 0,C 180,E1 -29109.819,E2 -29109.819} C_VEL
LIN {X 0,Y 66.89,Z 375.439,A -85,B 0,C 180,E1 -29117.351,E2 -29117.351} C_VEL
LIN {X 0,Y 74.431,Z 370.413,A -85,B 0,C 180,E1 -29123.382,E2 -29123.382} C_VEL
LIN {X 0,Y 82.563,Z 364.081,A -85,B 0,C 180,E1 -29128.349,E2 -29128.349} C_VEL
LIN {X 0,Y 91.196,Z 356.064,A -85,B 0,C 180,E1 -29132.574,E2 -29132.574} C_VEL
LIN {X 0,Y 100.017,Z 346.316,A -85,B 0,C 180,E1 -29135.995,E2 -29135.995} C_VEL
LIN {X 0,Y 107.746,Z 335.953,A -85,B 0,C 180,E1 -29138.359,E2 -29138.359} C_VEL
LIN {X 0,Y 113.967,Z 325.696,A -85,B 0,C 180,E1 -29140.125,E2 -29140.125} C_VEL
LIN {X 0,Y 119.428,Z 314.663,A -85,B 0,C 180,E1 -29141.453,E2 -29141.453} C_VEL
LIN {X 0,Y 123.907,Z 302.997,A -85,B 0,C 180,E1 -29142.49,E2 -29142.49} C_VEL
LIN {X 0,Y 127.315,Z 290.574,A -85,B 0,C 180,E1 -29143.293,E2 -29143.293} C_VEL
LIN {X 0,Y 129.435,Z 278.884,A -85,B 0,C 180,E1 -29143.762,E2 -29143.762} C_VEL
LIN {X 0,Y 129.472,Z 277.85,A -85,B 0,C 180,E1 -29143.949,E2 -29143.949} C_VEL
LIN {X 0,Y 128.109,Z 273.907,A -85,B 0,C 180,E1 -29147.324,E2 -29147.324} C_VEL
LIN {X 0,Y 127.051,Z 271.096,A -85,B 0,C 180,E1 -29150.648,E2 -29150.648} C_VEL
LIN {X 0,Y 126.567,Z 269.525,A -85,B 0,C 180,E1 -29152.823,E2 -29152.823} C_VEL
LIN {X 0,Y 125.976,Z 266.826,A -85,B 0,C 180,E1 -29159.183,E2 -29159.183} C_VEL
LIN {X 0,Y 125.975,Z 266.842,A -85,B 0,C 180,E1 -29160.385,E2 -29160.385} C_VEL
LIN {X 0,Y 126.714,Z 269.955,A -85,B 0,C 180,E1 -29167.419,E2 -29167.419} C_VEL
LIN {X 0,Y 127.846,Z 273.287,A -85,B 0,C 180,E1 -29171.494,E2 -29171.494} C_VEL
LIN {X 0,Y 129.283,Z 277.158,A -85,B 0,C 180,E1 -29175.065,E2 -29175.065} C_VEL
LIN {X 0,Y 129.546,Z 278.425,A -85,B 0,C 180,E1 -29175.739,E2 -29175.739} C_VEL
LIN {X 0,Y 127.485,Z 291.094,A -85,B 0,C 180,E1 -29176.205,E2 -29176.205} C_VEL
LIN {X 0,Y 124.223,Z 303.413,A -85,B 0,C 180,E1 -29176.828,E2 -29176.828} C_VEL
LIN {X 0,Y 119.722,Z 315.559,A -85,B 0,C 180,E1 -29177.686,E2 -29177.686} C_VEL
LIN {X 0,Y 114.184,Z 326.984,A -85,B 0,C 180,E1 -29178.854,E2 -29178.854} C_VEL
LIN {X 0,Y 106.976,Z 338.736,A -85,B 0,C 180,E1 -29180.576,E2 -29180.576} C_VEL
LIN {X 0,Y 99.102,Z 349.171,A -85,B 0,C 180,E1 -29182.789,E2 -29182.789} C_VEL
LIN {X 0,Y 91.464,Z 357.625,A -85,B 0,C 180,E1 -29185.46,E2 -29185.46} C_VEL
LIN {X 0,Y 82.646,Z 365.888,A -85,B 0,C 180,E1 -29189.347,E2 -29189.347} C_VEL
LIN {X 0,Y 73.955,Z 372.889,A -85,B 0,C 180,E1 -29194.531,E2 -29194.531} C_VEL
LIN {X 0,Y 65.585,Z 378.663,A -85,B 0,C 180,E1 -29201.396,E2 -29201.396} C_VEL
LIN {X 0,Y 58.99,Z 382.636,A -85,B 0,C 180,E1 -29209.056,E2 -29209.056} C_VEL
LIN {X 0,Y 53.645,Z 385.577,A -85,B 0,C 180,E1 -29218.392,E2 -29218.392} C_VEL
LIN {X 0,Y 49.342,Z 387.994,A -85,B 0,C 180,E1 -29233.445,E2 -29233.445} C_VEL
LIN {X 0,Y 48.478,Z 388.615,A -85,B 0,C 180,E1 -29241.66,E2 -29241.66} C_VEL
LIN {X 0,Y 48.471,Z 388.838,A -85,B 0,C 180,E1 -29249.996,E2 -29249.996} C_VEL
LIN {X 0,Y 48.488,Z 388.595,A -85,B 0,C 180,E1 -29258.329,E2 -29258.329} C_VEL
LIN {X 0,Y 49.364,Z 387.962,A -85,B 0,C 180,E1 -29266.539,E2 -29266.539} C_VEL
LIN {X 0,Y 51.084,Z 386.938,A -85,B 0,C 180,E1 -29274.371,E2 -29274.371} C_VEL
LIN {X 0,Y 53.641,Z 385.511,A -85,B 0,C 180,E1 -29281.601,E2 -29281.601} C_VEL
LIN {X 0,Y 58.985,Z 382.543,A -85,B 0,C 180,E1 -29290.939,E2 -29290.939} C_VEL
LIN {X 0,Y 65.582,Z 378.536,A -85,B 0,C 180,E1 -29298.597,E2 -29298.597} C_VEL
LIN {X 0,Y 73.254,Z 373.239,A -85,B 0,C 180,E1 -29304.993,E2 -29304.993} C_VEL
LIN {X 0,Y 81.232,Z 366.911,A -85,B 0,C 180,E1 -29309.896,E2 -29309.896} C_VEL
LIN {X 0,Y 89.955,Z 358.854,A -85,B 0,C 180,E1 -29313.95,E2 -29313.95} C_VEL
LIN {X 0,Y 97.548,Z 350.647,A -85,B 0,C 180,E1 -29316.714,E2 -29316.714} C_VEL
LIN {X 0,Y 105.372,Z 340.645,A -85,B 0,C 180,E1 -29319.02,E2 -29319.02} C_VEL
LIN {X 0,Y 112.554,Z 329.333,A -85,B 0,C 180,E1 -29320.8,E2 -29320.8} C_VEL
LIN {X 0,Y 118.2,Z 318.247,A -85,B 0,C 180,E1 -29322.044,E2 -29322.044} C_VEL
LIN {X 0,Y 122.98,Z 306.275,A -85,B 0,C 180,E1 -29322.966,E2 -29322.966} C_VEL
LIN {X 0,Y 126.638,Z 293.478,A -85,B 0,C 180,E1 -29323.66,E2 -29323.66} C_VEL
LIN {X 0,Y 128.958,Z 280.396,A -85,B 0,C 180,E1 -29324.188,E2 -29324.188} C_VEL
LIN {X 0,Y 129.187,Z 277.813,A -85,B 0,C 180,E1 -29324.419,E2 -29324.419} C_VEL
LIN {X 0,Y 128.299,Z 274.901,A -85,B 0,C 180,E1 -29326.538,E2 -29326.538} C_VEL
LIN {X 0,Y 127.053,Z 271.603,A -85,B 0,C 180,E1 -29330.046,E2 -29330.046} C_VEL
LIN {X 0,Y 126.271,Z 269.333,A -85,B 0,C 180,E1 -29333.208,E2 -29333.208} C_VEL
LIN {X 0,Y 125.698,Z 266.185,A -85,B 0,C 180,E1 -29340,E2 -29340} C_VEL
LIN {X 0,Y 125.685,Z 267.295,A -85,B 0,C 180,E1 -29342.834,E2 -29342.834} C_VEL
LIN {X 0,Y 126.498,Z 269.957,A -85,B 0,C 180,E1 -29348.386,E2 -29348.386} C_VEL
LIN {X 0,Y 127.712,Z 273.396,A -85,B 0,C 180,E1 -29352.514,E2 -29352.514} C_VEL
LIN {X 0,Y 129.112,Z 277.39,A -85,B 0,C 180,E1 -29355.996,E2 -29355.996} C_VEL
LIN {X 0,Y 129.239,Z 277.747,A -85,B 0,C 180,E1 -29356.28,E2 -29356.28} C_VEL
LIN {X 0,Y 127.165,Z 289.794,A -85,B 0,C 180,E1 -29356.789,E2 -29356.789} C_VEL
LIN {X 0,Y 126.203,Z 293.609,A -85,B 0,C 180,E1 -29356.874,E2 -29356.874} C_VEL
LIN {X 0,Y 123.574,Z 301.028,A -85,B 0,C 180,E1 -29356.478,E2 -29356.478} C_VEL
LIN {X 0,Y 117.816,Z 313.562,A -85,B 0,C 180,E1 -29355.562,E2 -29355.562} C_VEL
LIN {X 0,Y 115.235,Z 318.811,A -85,B 0,C 180,E1 -29355.786,E2 -29355.786} C_VEL
LIN {X 0,Y 109.363,Z 329.522,A -85,B 0,C 180,E1 -29357.086,E2 -29357.086} C_VEL
LIN {X 0,Y 102.125,Z 340.168,A -85,B 0,C 180,E1 -29358.882,E2 -29358.882} C_VEL
LIN {X 0,Y 94.242,Z 349.745,A -85,B 0,C 180,E1 -29361.232,E2 -29361.232} C_VEL
LIN {X 0,Y 85.769,Z 358.341,A -85,B 0,C 180,E1 -29364.396,E2 -29364.396} C_VEL
LIN {X 0,Y 76.189,Z 366.346,A -85,B 0,C 180,E1 -29368.806,E2 -29368.806} C_VEL
LIN {X 0,Y 67.669,Z 372.275,A -85,B 0,C 180,E1 -29373.82,E2 -29373.82} C_VEL
LIN {X 0,Y 59.85,Z 376.952,A -85,B 0,C 180,E1 -29380.253,E2 -29380.253} C_VEL
LIN {X 0,Y 52.961,Z 380.525,A -85,B 0,C 180,E1 -29388.438,E2 -29388.438} C_VEL
LIN {X 0,Y 49.038,Z 382.368,A -85,B 0,C 180,E1 -29395.028,E2 -29395.028} C_VEL
LIN {X 0,Y 45.855,Z 383.747,A -85,B 0,C 180,E1 -29402.631,E2 -29402.631} C_VEL
LIN {X 0,Y 42.049,Z 385.328,A -85,B 0,C 180,E1 -29420.384,E2 -29420.384} C_VEL
LIN {X 0,Y 41.637,Z 385.548,A -85,B 0,C 180,E1 -29430.005,E2 -29430.005} C_VEL
LIN {X 0,Y 42.05,Z 385.353,A -85,B 0,C 180,E1 -29439.626,E2 -29439.626} C_VEL
LIN {X 0,Y 45.846,Z 383.804,A -85,B 0,C 180,E1 -29457.385,E2 -29457.385} C_VEL
LIN {X 0,Y 49.01,Z 382.451,A -85,B 0,C 180,E1 -29465.006,E2 -29465.006} C_VEL
LIN {X 0,Y 55.094,Z 379.585,A -85,B 0,C 180,E1 -29474.561,E2 -29474.561} C_VEL
LIN {X 0,Y 62.293,Z 375.697,A -85,B 0,C 180,E1 -29482.167,E2 -29482.167} C_VEL
LIN {X 0,Y 70.429,Z 370.671,A -85,B 0,C 180,E1 -29488.021,E2 -29488.021} C_VEL
LIN {X 0,Y 79.067,Z 364.339,A -85,B 0,C 180,E1 -29492.735,E2 -29492.735} C_VEL
LIN {X 0,Y 88.044,Z 356.427,A -85,B 0,C 180,E1 -29496.63,E2 -29496.63} C_VEL
LIN {X 0,Y 97.343,Z 346.573,A -85,B 0,C 180,E1 -29499.818,E2 -29499.818} C_VEL
LIN {X 0,Y 105.336,Z 336.209,A -85,B 0,C 180,E1 -29501.948,E2 -29501.948} C_VEL
LIN {X 0,Y 111.761,Z 325.95,A -85,B 0,C 180,E1 -29503.536,E2 -29503.536} C_VEL
LIN {X 0,Y 117.968,Z 313.579,A -85,B 0,C 180,E1 -29504.87,E2 -29504.87} C_VEL
LIN {X 0,Y 122.356,Z 301.99,A -85,B 0,C 180,E1 -29505.761,E2 -29505.761} C_VEL
LIN {X 0,Y 125.767,Z 289.451,A -85,B 0,C 180,E1 -29506.457,E2 -29506.457} C_VEL
LIN {X 0,Y 127.153,Z 282.109,A -85,B 0,C 180,E1 -29506.821,E2 -29506.821} C_VEL
LIN {X 0,Y 126.102,Z 278.525,A -85,B 0,C 180,E1 -29510.577,E2 -29510.577} C_VEL
LIN {X 0,Y 125.53,Z 276.379,A -85,B 0,C 180,E1 -29513.571,E2 -29513.571} C_VEL
LIN {X 0,Y 125.107,Z 273.859,A -85,B 0,C 180,E1 -29520,E2 -29520} C_VEL
LIN {X 0,Y 125.684,Z 276.916,A -85,B 0,C 180,E1 -29526.824,E2 -29526.824} C_VEL
LIN {X 0,Y 126.503,Z 279.832,A -85,B 0,C 180,E1 -29530.402,E2 -29530.402} C_VEL
LIN {X 0,Y 127.248,Z 282.206,A -85,B 0,C 180,E1 -29532.763,E2 -29532.763} C_VEL
LIN {X 0,Y 124.975,Z 293.974,A -85,B 0,C 180,E1 -29533.205,E2 -29533.205} C_VEL
LIN {X 0,Y 121.324,Z 306.249,A -85,B 0,C 180,E1 -29533.798,E2 -29533.798} C_VEL
LIN {X 0,Y 116.228,Z 318.628,A -85,B 0,C 180,E1 -29534.649,E2 -29534.649} C_VEL
LIN {X 0,Y 110.44,Z 329.586,A -85,B 0,C 180,E1 -29535.737,E2 -29535.737} C_VEL
LIN {X 0,Y 103.051,Z 340.773,A -85,B 0,C 180,E1 -29537.291,E2 -29537.291} C_VEL
LIN {X 0,Y 94.968,Z 350.706,A -85,B 0,C 180,E1 -29539.34,E2 -29539.34} C_VEL
LIN {X 0,Y 85.52,Z 360.346,A -85,B 0,C 180,E1 -29542.4,E2 -29542.4} C_VEL
LIN {X 0,Y 76.418,Z 368.023,A -85,B 0,C 180,E1 -29546.269,E2 -29546.269} C_VEL
LIN {X 0,Y 66.398,Z 375.117,A -85,B 0,C 180,E1 -29552.134,E2 -29552.134} C_VEL
LIN {X 0,Y 58.536,Z 379.84,A -85,B 0,C 180,E1 -29558.697,E2 -29558.697} C_VEL
LIN {X 0,Y 51.619,Z 383.453,A -85,B 0,C 180,E1 -29567.092,E2 -29567.092} C_VEL
LIN {X 0,Y 47.713,Z 385.317,A -85,B 0,C 180,E1 -29573.895,E2 -29573.895} C_VEL
LIN {X 0,Y 42.561,Z 387.734,A -85,B 0,C 180,E1 -29590.711,E2 -29590.711} C_VEL
LIN {X 0,Y 41.447,Z 388.356,A -85,B 0,C 180,E1 -29600.232,E2 -29600.232} C_VEL
LIN {X 0,Y 41.357,Z 388.578,A -85,B 0,C 180,E1 -29609.995,E2 -29609.995} C_VEL
LIN {X 0,Y 41.456,Z 388.335,A -85,B 0,C 180,E1 -29619.755,E2 -29619.755} C_VEL
LIN {X 0,Y 42.579,Z 387.701,A -85,B 0,C 180,E1 -29629.27,E2 -29629.27} C_VEL
LIN {X 0,Y 44.684,Z 386.678,A -85,B 0,C 180,E1 -29638.148,E2 -29638.148} C_VEL
LIN {X 0,Y 47.709,Z 385.25,A -85,B 0,C 180,E1 -29646.097,E2 -29646.097} C_VEL
LIN {X 0,Y 53.798,Z 382.281,A -85,B 0,C 180,E1 -29655.924,E2 -29655.924} C_VEL
LIN {X 0,Y 61.105,Z 378.275,A -85,B 0,C 180,E1 -29663.613,E2 -29663.613} C_VEL
LIN {X 0,Y 70.468,Z 372.221,A -85,B 0,C 180,E1 -29670.471,E2 -29670.471} C_VEL
LIN {X 0,Y 79.387,Z 365.409,A -85,B 0,C 180,E1 -29675.143,E2 -29675.143} C_VEL
LIN {X 0,Y 88.629,Z 357.1,A -85,B 0,C 180,E1 -29678.698,E2 -29678.698} C_VEL
LIN {X 0,Y 96.561,Z 348.575,A -85,B 0,C 180,E1 -29681.107,E2 -29681.107} C_VEL
LIN {X 0,Y 104.669,Z 338.053,A -85,B 0,C 180,E1 -29683.091,E2 -29683.091} C_VEL
LIN {X 0,Y 111.253,Z 327.642,A -85,B 0,C 180,E1 -29684.432,E2 -29684.432} C_VEL
LIN {X 0,Y 116.884,Z 316.56,A -85,B 0,C 180,E1 -29685.478,E2 -29685.478} C_VEL
LIN {X 0,Y 121.58,Z 304.569,A -85,B 0,C 180,E1 -29686.254,E2 -29686.254} C_VEL
LIN {X 0,Y 125.217,Z 291.5,A -85,B 0,C 180,E1 -29686.849,E2 -29686.849} C_VEL
LIN {X 0,Y 126.934,Z 281.805,A -85,B 0,C 180,E1 -29687.306,E2 -29687.306} C_VEL
LIN {X 0,Y 125.857,Z 278.31,A -85,B 0,C 180,E1 -29690.964,E2 -29690.964} C_VEL
LIN {X 0,Y 125.162,Z 275.97,A -85,B 0,C 180,E1 -29694.361,E2 -29694.361} C_VEL
LIN {X 0,Y 124.816,Z 273.372,A -85,B 0,C 180,E1 -29700,E2 -29700} C_VEL
LIN {X 0,Y 125.389,Z 276.65,A -85,B 0,C 180,E1 -29707.448,E2 -29707.448} C_VEL
LIN {X 0,Y 126.366,Z 280.122,A -85,B 0,C 180,E1 -29711.631,E2 -29711.631} C_VEL
LIN {X 0,Y 126.877,Z 281.884,A -85,B 0,C 180,E1 -29713.306,E2 -29713.306} C_VEL
LIN {X 0,Y 124.177,Z 294.626,A -85,B 0,C 180,E1 -29713.892,E2 -29713.892} C_VEL
LIN {X 0,Y 120.411,Z 306.617,A -85,B 0,C 180,E1 -29714.679,E2 -29714.679} C_VEL
LIN {X 0,Y 115.235,Z 318.811,A -85,B 0,C 180,E1 -29715.786,E2 -29715.786} C_VEL
LIN {X 0,Y 112.454,Z 324.001,A -85,B 0,C 180,E1 -29716.058,E2 -29716.058} C_VEL
LIN {X 0,Y 106.865,Z 332.174,A -85,B 0,C 180,E1 -29715.667,E2 -29715.667} C_VEL
LIN {X 0,Y 100.65,Z 339.898,A -85,B 0,C 180,E1 -29715.33,E2 -29715.33} C_VEL
LIN {X 0,Y 96.877,Z 344.381,A -85,B 0,C 180,E1 -29715.792,E2 -29715.792} C_VEL
LIN {X 0,Y 88.697,Z 353.306,A -85,B 0,C 180,E1 -29718.051,E2 -29718.051} C_VEL
LIN {X 0,Y 79.213,Z 361.89,A -85,B 0,C 180,E1 -29721.325,E2 -29721.325} C_VEL
LIN {X 0,Y 69.985,Z 368.737,A -85,B 0,C 180,E1 -29725.347,E2 -29725.347} C_VEL
LIN {X 0,Y 61.08,Z 374.221,A -85,B 0,C 180,E1 -29730.357,E2 -29730.357} C_VEL
LIN {X 0,Y 52.88,Z 378.514,A -85,B 0,C 180,E1 -29737.122,E2 -29737.122} C_VEL
LIN {X 0,Y 47.872,Z 380.785,A -85,B 0,C 180,E1 -29742.782,E2 -29742.782} C_VEL
LIN {X 0,Y 43.415,Z 382.628,A -85,B 0,C 180,E1 -29749.652,E2 -29749.652} C_VEL
LIN {X 0,Y 39.68,Z 384.007,A -85,B 0,C 180,E1 -29757.911,E2 -29757.911} C_VEL
LIN {X 0,Y 35.088,Z 385.586,A -85,B 0,C 180,E1 -29778.452,E2 -29778.452} C_VEL
LIN {X 0,Y 34.564,Z 385.806,A -85,B 0,C 180,E1 -29790.006,E2 -29790.006} C_VEL
LIN {X 0,Y 35.089,Z 385.611,A -85,B 0,C 180,E1 -29801.56,E2 -29801.56} C_VEL
LIN {X 0,Y 39.673,Z 384.063,A -85,B 0,C 180,E1 -29822.109,E2 -29822.109} C_VEL
LIN {X 0,Y 43.39,Z 382.709,A -85,B 0,C 180,E1 -29830.388,E2 -29830.388} C_VEL
LIN {X 0,Y 50.28,Z 379.844,A -85,B 0,C 180,E1 -29840.25,E2 -29840.25} C_VEL
LIN {X 0,Y 58.203,Z 375.956,A -85,B 0,C 180,E1 -29847.704,E2 -29847.704} C_VEL
LIN {X 0,Y 66.937,Z 370.929,A -85,B 0,C 180,E1 -29853.188,E2 -29853.188} C_VEL
LIN {X 0,Y 76.075,Z 364.596,A -85,B 0,C 180,E1 -29857.497,E2 -29857.497} C_VEL
LIN {X 0,Y 85.161,Z 356.976,A -85,B 0,C 180,E1 -29860.9,E2 -29860.9} C_VEL
LIN {X 0,Y 93.509,Z 348.605,A -85,B 0,C 180,E1 -29863.394,E2 -29863.394} C_VEL
LIN {X 0,Y 101.702,Z 338.743,A -85,B 0,C 180,E1 -29865.346,E2 -29865.346} C_VEL
LIN {X 0,Y 109.129,Z 327.626,A -85,B 0,C 180,E1 -29866.926,E2 -29866.926} C_VEL
LIN {X 0,Y 115.582,Z 315.421,A -85,B 0,C 180,E1 -29868.105,E2 -29868.105} C_VEL
LIN {X 0,Y 120.255,Z 303.917,A -85,B 0,C 180,E1 -29868.912,E2 -29868.912} C_VEL
LIN {X 0,Y 123.845,Z 291.697,A -85,B 0,C 180,E1 -29869.547,E2 -29869.547} C_VEL
LIN {X 0,Y 124.955,Z 286.661,A -85,B 0,C 180,E1 -29869.779,E2 -29869.779} C_VEL
LIN {X 0,Y 124.429,Z 284.016,A -85,B 0,C 180,E1 -29873.106,E2 -29873.106} C_VEL
LIN {X 0,Y 124.199,Z 282.679,A -85,B 0,C 180,E1 -29875.537,E2 -29875.537} C_VEL
LIN {X 0,Y 124.141,Z 280.999,A -85,B 0,C 180,E1 -29880,E2 -29880} C_VEL
LIN {X 0,Y 124.444,Z 283.615,A -85,B 0,C 180,E1 -29885.875,E2 -29885.875} C_VEL
LIN {X 0,Y 125.046,Z 286.682,A -85,B 0,C 180,E1 -29889.707,E2 -29889.707} C_VEL
LIN {X 0,Y 122.403,Z 297.988,A -85,B 0,C 180,E1 -29890.184,E2 -29890.184} C_VEL
LIN {X 0,Y 117.888,Z 311.104,A -85,B 0,C 180,E1 -29890.777,E2 -29890.777} C_VEL
LIN {X 0,Y 112.096,Z 323.379,A -85,B 0,C 180,E1 -29891.58,E2 -29891.58} C_VEL
LIN {X 0,Y 105.358,Z 334.63,A -85,B 0,C 180,E1 -29892.684,E2 -29892.684} C_VEL
LIN {X 0,Y 97.831,Z 344.762,A -85,B 0,C 180,E1 -29894.107,E2 -29894.107} C_VEL
LIN {X 0,Y 89.578,Z 353.903,A -85,B 0,C 180,E1 -29896.029,E2 -29896.029} C_VEL
LIN {X 0,Y 79.847,Z 362.82,A -85,B 0,C 180,E1 -29898.875,E2 -29898.875} C_VEL
LIN {X 0,Y 70.447,Z 370.003,A -85,B 0,C 180,E1 -29902.655,E2 -29902.655} C_VEL
LIN {X 0,Y 59.99,Z 376.552,A -85,B 0,C 180,E1 -29908.515,E2 -29908.515} C_VEL
LIN {X 0,Y 51.667,Z 380.89,A -85,B 0,C 180,E1 -29915.293,E2 -29915.293} C_VEL
LIN {X 0,Y 46.646,Z 383.194,A -85,B 0,C 180,E1 -29921.115,E2 -29921.115} C_VEL
LIN {X 0,Y 42.156,Z 385.057,A -85,B 0,C 180,E1 -29928.169,E2 -29928.169} C_VEL
LIN {X 0,Y 35.922,Z 387.475,A -85,B 0,C 180,E1 -29946.959,E2 -29946.959} C_VEL
LIN {X 0,Y 34.465,Z 388.096,A -85,B 0,C 180,E1 -29958.228,E2 -29958.228} C_VEL
LIN {X 0,Y 34.262,Z 388.319,A -85,B 0,C 180,E1 -29969.994,E2 -29969.994} C_VEL
LIN {X 0,Y 34.473,Z 388.076,A -85,B 0,C 180,E1 -29981.757,E2 -29981.757} C_VEL
LIN {X 0,Y 35.936,Z 387.441,A -85,B 0,C 180,E1 -29993.019,E2 -29993.019} C_VEL
LIN {X 0,Y 38.548,Z 386.417,A -85,B 0,C 180,E1 -30003.151,E2 -30003.151} C_VEL
LIN {X 0,Y 42.151,Z 384.988,A -85,B 0,C 180,E1 -30011.823,E2 -30011.823} C_VEL
LIN {X 0,Y 49.104,Z 382.02,A -85,B 0,C 180,E1 -30021.915,E2 -30021.915} C_VEL
LIN {X 0,Y 57.167,Z 378.014,A -85,B 0,C 180,E1 -30029.371,E2 -30029.371} C_VEL
LIN {X 0,Y 67.236,Z 371.959,A -85,B 0,C 180,E1 -30035.774,E2 -30035.774} C_VEL
LIN {X 0,Y 76.659,Z 365.146,A -85,B 0,C 180,E1 -30039.992,E2 -30039.992} C_VEL
LIN {X 0,Y 86.302,Z 356.838,A -85,B 0,C 180,E1 -30043.097,E2 -30043.097} C_VEL
LIN {X 0,Y 94.5,Z 348.313,A -85,B 0,C 180,E1 -30045.185,E2 -30045.185} C_VEL
LIN {X 0,Y 102.825,Z 337.789,A -85,B 0,C 180,E1 -30046.888,E2 -30046.888} C_VEL
LIN {X 0,Y 109.558,Z 327.378,A -85,B 0,C 180,E1 -30048.019,E2 -30048.019} C_VEL
LIN {X 0,Y 115.241,Z 316.439,A -85,B 0,C 180,E1 -30048.882,E2 -30048.882} C_VEL
LIN {X 0,Y 120.279,Z 303.711,A -85,B 0,C 180,E1 -30049.583,E2 -30049.583} C_VEL
LIN {X 0,Y 123.98,Z 290.418,A -85,B 0,C 180,E1 -30050.082,E2 -30050.082} C_VEL
LIN {X 0,Y 124.775,Z 286.368,A -85,B 0,C 180,E1 -30050.272,E2 -30050.272} C_VEL
LIN {X 0,Y 124.084,Z 282.977,A -85,B 0,C 180,E1 -30054.719,E2 -30054.719} C_VEL
LIN {X 0,Y 123.848,Z 280.595,A -85,B 0,C 180,E1 -30060,E2 -30060} C_VEL
LIN {X 0,Y 124.089,Z 283.168,A -85,B 0,C 180,E1 -30066.3,E2 -30066.3} C_VEL
LIN {X 0,Y 124.672,Z 286.382,A -85,B 0,C 180,E1 -30070.321,E2 -30070.321} C_VEL
LIN {X 0,Y 121.657,Z 298.549,A -85,B 0,C 180,E1 -30070.88,E2 -30070.88} C_VEL
LIN {X 0,Y 117.291,Z 310.738,A -85,B 0,C 180,E1 -30071.643,E2 -30071.643} C_VEL
LIN {X 0,Y 112.487,Z 321.05,A -85,B 0,C 180,E1 -30072.533,E2 -30072.533} C_VEL
LIN {X 0,Y 105.834,Z 332.359,A -85,B 0,C 180,E1 -30073.8,E2 -30073.8} C_VEL
LIN {X 0,Y 98.418,Z 342.546,A -85,B 0,C 180,E1 -30075.426,E2 -30075.426} C_VEL
LIN {X 0,Y 96.877,Z 344.381,A -85,B 0,C 180,E1 -30075.792,E2 -30075.792} C_VEL
LIN {X 0,Y 92.933,Z 348.716,A -85,B 0,C 180,E1 -30076.358,E2 -30076.358} C_VEL
LIN {X 0,Y 85.612,Z 355.419,A -85,B 0,C 180,E1 -30076.4,E2 -30076.4} C_VEL
LIN {X 0,Y 77.833,Z 361.549,A -85,B 0,C 180,E1 -30076.61,E2 -30076.61} C_VEL
LIN {X 0,Y 73.196,Z 364.942,A -85,B 0,C 180,E1 -30077.635,E2 -30077.635} C_VEL
LIN {X 0,Y 64.075,Z 370.992,A -85,B 0,C 180,E1 -30081.213,E2 -30081.213} C_VEL
LIN {X 0,Y 54.763,Z 376.063,A -85,B 0,C 180,E1 -30086.07,E2 -30086.07} C_VEL
LIN {X 0,Y 46.09,Z 379.99,A -85,B 0,C 180,E1 -30093.011,E2 -30093.011} C_VEL
LIN {X 0,Y 38.287,Z 382.887,A -85,B 0,C 180,E1 -30102.766,E2 -30102.766} C_VEL
LIN {X 0,Y 33.881,Z 384.266,A -85,B 0,C 180,E1 -30111.525,E2 -30111.525} C_VEL
LIN {X 0,Y 28.17,Z 385.846,A -85,B 0,C 180,E1 -30135.561,E2 -30135.561} C_VEL
LIN {X 0,Y 27.48,Z 386.065,A -85,B 0,C 180,E1 -30150.008,E2 -30150.008} C_VEL
LIN {X 0,Y 28.172,Z 385.87,A -85,B 0,C 180,E1 -30164.454,E2 -30164.454} C_VEL
LIN {X 0,Y 33.875,Z 384.322,A -85,B 0,C 180,E1 -30188.499,E2 -30188.499} C_VEL
LIN {X 0,Y 38.268,Z 382.967,A -85,B 0,C 180,E1 -30197.282,E2 -30197.282} C_VEL
LIN {X 0,Y 46.066,Z 380.102,A -85,B 0,C 180,E1 -30207.052,E2 -30207.052} C_VEL
LIN {X 0,Y 54.736,Z 376.214,A -85,B 0,C 180,E1 -30214.005,E2 -30214.005} C_VEL
LIN {X 0,Y 64.049,Z 371.186,A -85,B 0,C 180,E1 -30218.865,E2 -30218.865} C_VEL
LIN {X 0,Y 73.648,Z 364.854,A -85,B 0,C 180,E1 -30222.613,E2 -30222.613} C_VEL
LIN {X 0,Y 83.437,Z 356.94,A -85,B 0,C 180,E1 -30225.615,E2 -30225.615} C_VEL
LIN {X 0,Y 93.403,Z 347.085,A -85,B 0,C 180,E1 -30228.014,E2 -30228.014} C_VEL
LIN {X 0,Y 101.835,Z 336.72,A -85,B 0,C 180,E1 -30229.566,E2 -30229.566} C_VEL
LIN {X 0,Y 108.598,Z 326.458,A -85,B 0,C 180,E1 -30230.726,E2 -30230.726} C_VEL
LIN {X 0,Y 114.814,Z 314.675,A -85,B 0,C 180,E1 -30231.653,E2 -30231.653} C_VEL
LIN {X 0,Y 119.537,Z 302.87,A -85,B 0,C 180,E1 -30232.329,E2 -30232.329} C_VEL
LIN {X 0,Y 122.86,Z 291.405,A -85,B 0,C 180,E1 -30232.908,E2 -30232.908} C_VEL
LIN {X 0,Y 122.738,Z 289.779,A -85,B 0,C 180,E1 -30235.484,E2 -30235.484} C_VEL
LIN {X 0,Y 122.837,Z 288.09,A -85,B 0,C 180,E1 -30240,E2 -30240} C_VEL
LIN {X 0,Y 122.874,Z 290.39,A -85,B 0,C 180,E1 -30245.127,E2 -30245.127} C_VEL
LIN {X 0,Y 122.973,Z 291.472,A -85,B 0,C 180,E1 -30246.631,E2 -30246.631} C_VEL
LIN {X 0,Y 119.831,Z 302.572,A -85,B 0,C 180,E1 -30247.016,E2 -30247.016} C_VEL
LIN {X 0,Y 115.225,Z 314.427,A -85,B 0,C 180,E1 -30247.538,E2 -30247.538} C_VEL
LIN {X 0,Y 109.175,Z 326.219,A -85,B 0,C 180,E1 -30248.204,E2 -30248.204} C_VEL
LIN {X 0,Y 101.463,Z 337.969,A -85,B 0,C 180,E1 -30249.225,E2 -30249.225} C_VEL
LIN {X 0,Y 92.948,Z 348.402,A -85,B 0,C 180,E1 -30250.585,E2 -30250.585} C_VEL
LIN {X 0,Y 82.837,Z 358.344,A -85,B 0,C 180,E1 -30252.656,E2 -30252.656} C_VEL
LIN {X 0,Y 72.89,Z 366.351,A -85,B 0,C 180,E1 -30255.37,E2 -30255.37} C_VEL
LIN {X 0,Y 63.211,Z 372.775,A -85,B 0,C 180,E1 -30259.073,E2 -30259.073} C_VEL
LIN {X 0,Y 53.878,Z 377.885,A -85,B 0,C 180,E1 -30264.056,E2 -30264.056} C_VEL
LIN {X 0,Y 45.063,Z 381.857,A -85,B 0,C 180,E1 -30270.925,E2 -30270.925} C_VEL
LIN {X 0,Y 37.144,Z 384.797,A -85,B 0,C 180,E1 -30280.806,E2 -30280.806} C_VEL
LIN {X 0,Y 29.487,Z 387.214,A -85,B 0,C 180,E1 -30301.523,E2 -30301.523} C_VEL
LIN {X 0,Y 27.531,Z 387.836,A -85,B 0,C 180,E1 -30315.203,E2 -30315.203} C_VEL
LIN {X 0,Y 27.148,Z 388.059,A -85,B 0,C 180,E1 -30329.992,E2 -30329.992} C_VEL
LIN {X 0,Y 27.538,Z 387.815,A -85,B 0,C 180,E1 -30344.778,E2 -30344.778} C_VEL
LIN {X 0,Y 32.804,Z 386.156,A -85,B 0,C 180,E1 -30369.986,E2 -30369.986} C_VEL
LIN {X 0,Y 37.139,Z 384.727,A -85,B 0,C 180,E1 -30379.186,E2 -30379.186} C_VEL
LIN {X 0,Y 45.057,Z 381.759,A -85,B 0,C 180,E1 -30389.071,E2 -30389.071} C_VEL
LIN {X 0,Y 56.035,Z 376.616,A -85,B 0,C 180,E1 -30397.274,E2 -30397.274} C_VEL
LIN {X 0,Y 66.401,Z 370.58,A -85,B 0,C 180,E1 -30402.271,E2 -30402.271} C_VEL
LIN {X 0,Y 76.175,Z 363.646,A -85,B 0,C 180,E1 -30405.623,E2 -30405.623} C_VEL
LIN {X 0,Y 86.184,Z 354.975,A -85,B 0,C 180,E1 -30408.097,E2 -30408.097} C_VEL
LIN {X 0,Y 94.646,Z 346.097,A -85,B 0,C 180,E1 -30409.684,E2 -30409.684} C_VEL
LIN {X 0,Y 102.304,Z 336.35,A -85,B 0,C 180,E1 -30410.921,E2 -30410.921} C_VEL
LIN {X 0,Y 109.168,Z 325.68,A -85,B 0,C 180,E1 -30411.793,E2 -30411.793} C_VEL
LIN {X 0,Y 115.104,Z 313.908,A -85,B 0,C 180,E1 -30412.492,E2 -30412.492} C_VEL
LIN {X 0,Y 120.007,Z 300.997,A -85,B 0,C 180,E1 -30413.036,E2 -30413.036} C_VEL
LIN {X 0,Y 122.707,Z 291.162,A -85,B 0,C 180,E1 -30413.356,E2 -30413.356} C_VEL
LIN {X 0,Y 122.513,Z 289.361,A -85,B 0,C 180,E1 -30416.3,E2 -30416.3} C_VEL
LIN {X 0,Y 122.558,Z 287.741,A -85,B 0,C 180,E1 -30420,E2 -30420} C_VEL
LIN {X 0,Y 122.516,Z 289.927,A -85,B 0,C 180,E1 -30425.555,E2 -30425.555} C_VEL
LIN {X 0,Y 122.583,Z 291.171,A -85,B 0,C 180,E1 -30427.225,E2 -30427.225} C_VEL
LIN {X 0,Y 119.063,Z 303.274,A -85,B 0,C 180,E1 -30427.797,E2 -30427.797} C_VEL
LIN {X 0,Y 114.223,Z 315.185,A -85,B 0,C 180,E1 -30428.472,E2 -30428.472} C_VEL
LIN {X 0,Y 107.764,Z 327.299,A -85,B 0,C 180,E1 -30429.478,E2 -30429.478} C_VEL
LIN {X 0,Y 101.002,Z 337.408,A -85,B 0,C 180,E1 -30430.64,E2 -30430.64} C_VEL
LIN {X 0,Y 93.424,Z 346.699,A -85,B 0,C 180,E1 -30432.068,E2 -30432.068} C_VEL
LIN {X 0,Y 85.106,Z 355.155,A -85,B 0,C 180,E1 -30434.016,E2 -30434.016} C_VEL
LIN {X 0,Y 75.302,Z 363.374,A -85,B 0,C 180,E1 -30436.946,E2 -30436.946} C_VEL
LIN {X 0,Y 73.196,Z 364.942,A -85,B 0,C 180,E1 -30437.635,E2 -30437.635} C_VEL
LIN {X 0,Y 68.426,Z 368.143,A -85,B 0,C 180,E1 -30438.81,E2 -30438.81} C_VEL
LIN {X 0,Y 59.767,Z 372.889,A -85,B 0,C 180,E1 -30439.534,E2 -30439.534} C_VEL
LIN {X 0,Y 50.789,Z 376.986,A -85,B 0,C 180,E1 -30440.597,E2 -30440.597} C_VEL
LIN {X 0,Y 45.598,Z 379.084,A -85,B 0,C 180,E1 -30442.835,E2 -30442.835} C_VEL
LIN {X 0,Y 39.615,Z 381.306,A -85,B 0,C 180,E1 -30447.51,E2 -30447.51} C_VEL
LIN {X 0,Y 33.878,Z 383.146,A -85,B 0,C 180,E1 -30453.935,E2 -30453.935} C_VEL
LIN {X 0,Y 24.324,Z 385.506,A -85,B 0,C 180,E1 -30474.71,E2 -30474.71} C_VEL
LIN {X 0,Y 21.385,Z 386.104,A -85,B 0,C 180,E1 -30490.825,E2 -30490.825} C_VEL
LIN {X 0,Y 20.384,Z 386.324,A -85,B 0,C 180,E1 -30510.01,E2 -30510.01} C_VEL
LIN {X 0,Y 21.388,Z 386.128,A -85,B 0,C 180,E1 -30529.194,E2 -30529.194} C_VEL
LIN {X 0,Y 28.656,Z 384.581,A -85,B 0,C 180,E1 -30557.382,E2 -30557.382} C_VEL
LIN {X 0,Y 33.847,Z 383.226,A -85,B 0,C 180,E1 -30566.166,E2 -30566.166} C_VEL
LIN {X 0,Y 42.625,Z 380.36,A -85,B 0,C 180,E1 -30575.082,E2 -30575.082} C_VEL
LIN {X 0,Y 52.017,Z 376.472,A -85,B 0,C 180,E1 -30581.053,E2 -30581.053} C_VEL
LIN {X 0,Y 61.846,Z 371.444,A -85,B 0,C 180,E1 -30585.008,E2 -30585.008} C_VEL
LIN {X 0,Y 71.845,Z 365.111,A -85,B 0,C 180,E1 -30588.031,E2 -30588.031} C_VEL
LIN {X 0,Y 81.628,Z 357.489,A -85,B 0,C 180,E1 -30590.349,E2 -30590.349} C_VEL
